C03632=1072.520,220.619,417.871,174.022,27.766,154.945
C03633=1072.515,220.371,417.896,174.019,27.761,154.944
C03634=1072.509,220.122,417.922,174.017,27.758,154.944
C03635=1072.503,219.873,417.948,174.015,27.754,154.943
C03636=1072.497,219.625,417.973,174.012,27.750,154.943
C03637=1072.491,219.377,417.999,174.010,27.746,154.942
C03638=1072.485,219.128,418.025,174.009,27.743,154.941
C03639=1072.479,218.879,418.050,174.006,27.738,154.941
C03640=1072.473,218.630,418.076,174.004,27.734,154.940
C03641=1072.468,218.382,418.101,174.002,27.731,154.940
C03642=1072.462,218.133,418.127,173.999,27.727,154.939
C03643=1072.456,217.885,418.152,173.998,27.723,154.938
C03644=1072.450,217.636,418.178,173.996,27.719,154.938
C03645=1072.444,217.387,418.204,173.994,27.715,154.937
C03646=1072.439,217.139,418.229,173.991,27.711,154.936
C03647=1072.433,216.890,418.254,173.989,27.707,154.936
C03648=1072.427,216.641,418.280,173.987,27.703,154.935
C03649=1072.421,216.393,418.305,173.985,27.699,154.935
C03650=1072.415,216.144,418.331,173.983,27.695,154.934
C03651=1072.410,215.896,418.356,173.981,27.692,154.933
C03652=1072.404,215.647,418.382,173.978,27.688,154.933
C03653=1072.398,215.398,418.407,173.976,27.684,154.932
C03654=1072.392,215.149,418.433,173.975,27.680,154.931
C03655=1072.386,214.901,418.458,173.972,27.676,154.931
C03656=1072.381,214.652,418.482,173.970,27.672,154.930
C03657=1072.375,214.403,418.508,173.968,27.668,154.930
C03658=1072.369,214.154,418.534,173.965,27.664,154.929
C03659=1072.363,213.906,418.559,173.964,27.660,154.928
C03660=1072.358,213.657,418.585,173.962,27.656,154.928
C03661=1072.352,213.409,418.610,173.960,27.652,154.927
C03662=1072.346,213.161,418.635,173.957,27.648,154.926
C03663=1072.340,212.912,418.660,173.956,27.645,154.926
C03664=1072.335,212.663,418.685,173.954,27.641,154.925
C03665=1072.328,212.414,418.711,173.951,27.637,154.925
C03666=1072.323,212.166,418.736,173.949,27.633,154.924
C03667=1072.317,211.917,418.760,173.947,27.629,154.923
C03668=1072.311,211.668,418.786,173.945,27.625,154.923
C03669=1072.306,211.420,418.811,173.943,27.621,154.922
C03670=1072.300,211.171,418.837,173.941,27.617,154.922
C03671=1072.294,210.922,418.861,173.939,27.613,154.921
C03672=1072.288,210.673,418.887,173.937,27.609,154.920
C03673=1072.282,210.425,418.912,173.935,27.606,154.920
C03674=1072.276,210.176,418.936,173.933,27.602,154.919
C03675=1072.270,209.927,418.962,173.930,27.598,154.918
C03676=1072.264,209.679,418.987,173.928,27.593,154.918
C03677=1072.258,209.430,419.011,173.927,27.590,154.917
C03678=1072.249,209.010,419.054,173.923,27.583,154.916
C03679=1072.239,208.591,419.096,173.919,27.577,154.915
C03680=1072.229,208.171,419.138,173.916,27.570,154.914
C03681=1072.220,207.751,419.180,173.912,27.563,154.913
C03682=1072.195,206.710,419.281,173.782,27.496,154.911
C03683=1072.190,206.461,419.306,173.780,27.493,154.911
C03684=1072.184,206.212,419.330,173.778,27.490,154.911
C03685=1072.178,205.964,419.354,173.776,27.487,154.910
C03686=1072.173,205.715,419.378,173.773,27.484,154.910
C03687=1072.167,205.466,419.403,173.771,27.480,154.909
C03688=1072.161,205.217,419.427,173.769,27.477,154.909
C03689=1072.155,204.969,419.451,173.767,27.475,154.909
C03690=1072.150,204.720,419.475,173.765,27.472,154.908
C03691=1072.144,204.471,419.500,173.762,27.469,154.908
C03692=1072.139,204.222,419.524,173.760,27.465,154.907
C03693=1072.133,203.974,419.548,173.758,27.463,154.907
C03694=1072.127,203.724,419.572,173.756,27.460,154.907
C03695=1072.122,203.476,419.596,173.753,27.457,154.906
C03696=1072.116,203.227,419.619,173.751,27.454,154.906
C03697=1072.111,202.979,419.644,173.749,27.451,154.905
C03698=1072.105,202.729,419.668,173.747,27.448,154.905
C03699=1072.099,202.481,419.693,173.745,27.444,154.905
C03700=1072.094,202.232,419.716,173.742,27.441,154.904
C03701=1072.088,201.983,419.740,173.741,27.439,154.904
C03702=1072.082,201.734,419.764,173.738,27.436,154.903
C03703=1072.076,201.486,419.788,173.736,27.433,154.903
C03704=1072.070,201.238,419.812,173.733,27.430,154.903
C03705=1072.065,200.988,419.836,173.732,27.427,154.902
C03706=1072.059,200.739,419.859,173.729,27.424,154.902
C03707=1072.053,200.491,419.883,173.727,27.421,154.902
C03708=1072.047,200.241,419.907,173.724,27.418,154.901
C03709=1072.041,199.993,419.931,173.723,27.416,154.901
C03710=1072.036,199.744,419.955,173.720,27.413,154.900
C03711=1072.030,199.495,419.978,173.718,27.410,154.900
C03712=1072.024,199.246,420.002,173.716,27.407,154.900
C03713=1072.018,198.998,420.026,173.714,27.404,154.899
C03714=1072.013,198.749,420.050,173.712,27.401,154.899
C03715=1072.007,198.500,420.073,173.709,27.398,154.898
C03716=1072.001,198.251,420.097,173.707,27.395,154.898
C03717=1071.996,198.002,420.121,173.705,27.393,154.898
C03718=1071.989,197.754,420.144,173.703,27.390,154.897
C03719=1071.984,197.505,420.168,173.700,27.387,154.897
C03720=1071.978,197.256,420.192,173.699,27.384,154.897
C03721=1071.972,197.007,420.216,173.696,27.381,154.896
C03722=1071.967,196.758,420.239,173.694,27.378,154.896
C03723=1071.961,196.510,420.263,173.692,27.375,154.895
C03724=1071.956,196.261,420.286,173.690,27.372,154.895
C03725=1071.950,196.012,420.310,173.688,27.369,154.895
C03726=1071.943,195.763,420.333,173.685,27.366,154.894
C03727=1071.938,195.514,420.358,173.684,27.364,154.894
C03728=1071.932,195.265,420.381,173.681,27.361,154.893
C03729=1071.927,195.017,420.405,173.679,27.358,154.893
C03730=1071.921,194.768,420.428,173.677,27.355,154.893
C03731=1071.915,194.520,420.451,173.675,27.352,154.892
C03732=1071.910,194.270,420.475,173.672,27.349,154.892
C03733=1071.904,194.021,420.499,173.671,27.346,154.892
C03734=1071.898,193.773,420.522,173.668,27.343,154.891
C03735=1071.893,193.523,420.546,173.666,27.340,154.891
C03736=1071.887,193.275,420.569,173.664,27.337,154.890
C03737=1071.881,193.026,420.592,173.662,27.334,154.890
C03738=1071.876,192.778,420.616,173.660,27.331,154.890
C03739=1071.870,192.529,420.639,173.658,27.328,154.889
C03740=1071.864,192.280,420.662,173.656,27.325,154.889
C03741=1071.859,192.031,420.687,173.653,27.323,154.888
C03742=1071.853,191.782,420.709,173.652,27.320,154.888
C03743=1071.847,191.501,420.736,173.649,27.317,154.888
C03744=1071.841,191.219,420.762,173.647,27.314,154.887
C03745=1071.834,190.938,420.789,173.645,27.310,154.887
C03746=1071.828,190.656,420.816,173.642,27.307,154.886
C03747=1071.822,190.407,420.839,173.640,27.304,154.886
C03748=1071.817,190.158,420.862,173.637,27.301,154.886
C03749=1071.811,189.909,420.885,173.636,27.298,154.885
C03750=1071.805,189.661,420.909,173.633,27.295,154.885
C03751=1071.800,189.411,420.932,173.631,27.292,154.884
C03752=1071.795,189.162,420.955,173.629,27.289,154.884
C03753=1071.789,188.914,420.978,173.627,27.286,154.884
C03754=1071.783,188.665,421.002,173.625,27.283,154.883
C03755=1071.778,188.416,421.025,173.623,27.281,154.883
C03756=1071.772,188.167,421.048,173.621,27.278,154.882
C03757=1071.766,187.918,421.071,173.619,27.275,154.882
C03758=1071.761,187.669,421.095,173.617,27.272,154.882
C03759=1071.755,187.421,421.119,173.614,27.269,154.881
C03760=1071.750,187.172,421.141,173.613,27.267,154.881
C03761=1071.744,186.923,421.164,173.610,27.263,154.881
C03762=1071.739,186.674,421.188,173.608,27.260,154.880
C03763=1071.733,186.425,421.211,173.606,27.258,154.880
C03764=1071.728,186.176,421.234,173.604,27.255,154.879
C03765=1071.722,185.927,421.257,173.602,27.252,154.879
C03766=1071.717,185.678,421.280,173.600,27.249,154.879
C03767=1071.711,185.429,421.303,173.598,27.246,154.878
C03768=1071.705,185.180,421.326,173.596,27.243,154.878
C03769=1071.700,184.931,421.349,173.594,27.240,154.877
C03770=1071.694,184.683,421.372,173.592,27.237,154.877
C03771=1071.688,184.433,421.395,173.590,27.234,154.877
C03772=1071.682,184.185,421.418,173.587,27.232,154.876
C03773=1071.677,183.936,421.441,173.586,27.229,154.876
C03774=1071.671,183.687,421.464,173.583,27.226,154.875
C03775=1071.665,183.438,421.487,173.582,27.224,154.875
C03776=1071.659,183.189,421.510,173.579,27.221,154.875
C03777=1071.653,182.940,421.532,173.577,27.218,154.874
C03778=1071.647,182.691,421.555,173.575,27.215,154.874
C03779=1071.642,182.443,421.578,173.573,27.212,154.874
C03780=1071.636,182.194,421.601,173.571,27.210,154.873
C03781=1071.630,181.945,421.624,173.569,27.207,154.873
C03782=1071.624,181.696,421.646,173.567,27.204,154.873
C03783=1071.618,181.447,421.669,173.565,27.201,154.872
C03784=1071.612,181.198,421.691,173.563,27.198,154.872
C03785=1071.607,180.949,421.714,173.561,27.196,154.872
C03786=1071.602,180.701,421.737,173.559,27.193,154.871
C03787=1071.595,180.452,421.759,173.557,27.190,154.871
C03788=1071.589,180.203,421.782,173.555,27.188,154.871
C03789=1071.584,179.954,421.805,173.552,27.185,154.870
C03790=1071.578,179.705,421.827,173.551,27.182,154.870
C03791=1071.573,179.456,421.850,173.548,27.179,154.869
C03792=1071.566,179.207,421.873,173.547,27.177,154.869
C03793=1071.560,178.958,421.896,173.544,27.174,154.869
C03794=1071.555,178.709,421.919,173.543,27.171,154.868
C03795=1071.549,178.460,421.941,173.540,27.168,154.868
C03796=1071.543,178.211,421.963,173.539,27.166,154.868
C03797=1071.537,177.962,421.986,173.536,27.163,154.867
C03798=1071.532,177.714,422.008,173.534,27.160,154.867
C03799=1071.526,177.465,422.031,173.532,27.157,154.867
C03800=1071.520,177.216,422.053,173.530,27.154,154.866
C03801=1071.514,176.967,422.076,173.529,27.152,154.866
C03802=1071.509,176.718,422.098,173.526,27.148,154.865
C03803=1071.503,176.469,422.121,173.525,27.146,154.865
C03804=1071.497,176.220,422.144,173.522,27.143,154.865
C03805=1071.492,175.971,422.166,173.521,27.140,154.864
C03806=1071.486,175.723,422.189,173.518,27.137,154.864
C03807=1071.479,175.441,422.214,173.516,27.134,154.864
C03808=1071.473,175.158,422.239,173.513,27.131,154.863
C03809=1071.466,174.877,422.265,173.512,27.129,154.863
C03810=1071.460,174.595,422.290,173.510,27.125,154.862
C03811=1071.454,174.345,422.312,173.507,27.122,154.862
C03812=1071.448,174.096,422.335,173.506,27.120,154.862
C03813=1071.444,173.847,422.357,173.503,27.117,154.861
C03814=1071.437,173.599,422.380,173.502,27.114,154.861
C03815=1071.431,173.350,422.403,173.499,27.111,154.861
C03816=1071.426,173.100,422.425,173.498,27.109,154.860
C03817=1071.420,172.852,422.447,173.495,27.106,154.860
C03818=1071.415,172.603,422.469,173.494,27.103,154.859
C03819=1071.409,172.354,422.492,173.491,27.100,154.859
C03820=1071.403,172.105,422.514,173.490,27.097,154.859
C03821=1071.398,171.857,422.536,173.488,27.094,154.858
C03822=1071.392,171.607,422.558,173.486,27.092,154.858
C03823=1071.386,171.359,422.581,173.484,27.089,154.858
C03824=1071.380,171.109,422.603,173.482,27.086,154.857
C03825=1071.375,170.860,422.625,173.480,27.083,154.857
C03826=1071.369,170.612,422.647,173.478,27.081,154.856
C03827=1071.364,170.362,422.669,173.476,27.078,154.856
C03828=1071.358,170.113,422.692,173.474,27.075,154.856
C03829=1071.352,169.865,422.714,173.472,27.072,154.855
C03830=1071.347,169.616,422.737,173.470,27.069,154.855
C03831=1071.341,169.366,422.759,173.468,27.066,154.855
C03832=1071.336,169.118,422.780,173.466,27.064,154.854
C03833=1071.330,168.869,422.803,173.464,27.061,154.854
C03834=1071.324,168.619,422.825,173.463,27.058,154.853
C03835=1071.319,168.371,422.846,173.460,27.055,154.853
C03836=1071.313,168.122,422.869,173.459,27.052,154.853
C03837=1071.308,167.872,422.892,173.456,27.050,154.852
C03838=1071.302,167.624,422.913,173.455,27.047,154.852
C03839=1071.296,167.375,422.936,173.452,27.044,154.852
C03840=1071.290,167.126,422.958,173.451,27.041,154.851
C03841=1071.285,166.877,422.979,173.448,27.038,154.851
C03842=1071.280,166.628,423.002,173.447,27.036,154.851
C03843=1071.274,166.380,423.024,173.445,27.033,154.850
C03844=1071.269,166.130,423.046,173.443,27.030,154.850
C03845=1071.263,165.881,423.067,173.442,27.027,154.849
C03846=1071.258,165.632,423.089,173.439,27.024,154.849
C03847=1071.252,165.383,423.112,173.438,27.022,154.849
C03848=1071.246,165.135,423.134,173.435,27.019,154.848
C03849=1071.241,164.885,423.156,173.434,27.016,154.848
C03850=1071.235,164.636,423.177,173.431,27.013,154.848
C03851=1071.230,164.387,423.199,173.430,27.010,154.847
C03852=1071.224,164.138,423.222,173.428,27.008,154.847
C03853=1071.219,163.890,423.243,173.426,27.005,154.846
C03854=1071.213,163.640,423.266,173.424,27.002,154.846
C03855=1071.208,163.392,423.287,173.422,26.999,154.846
C03856=1071.202,163.142,423.309,173.421,26.997,154.845
C03857=1071.197,162.894,423.330,173.418,26.994,154.845
C03858=1071.191,162.645,423.353,173.417,26.991,154.844
C03859=1071.186,162.395,423.376,173.415,26.988,154.844
C03860=1071.180,162.147,423.397,173.413,26.985,154.844
C03861=1071.175,161.897,423.419,173.411,26.983,154.843
C03862=1071.169,161.649,423.440,173.409,26.980,154.843
C03863=1071.164,161.399,423.463,173.407,26.977,154.843
C03864=1071.158,161.151,423.484,173.405,26.974,154.842
C03865=1071.152,160.902,423.506,173.403,26.972,154.842
C03866=1071.147,160.653,423.527,173.402,26.969,154.841
C03867=1071.141,160.404,423.549,173.400,26.966,154.841
C03868=1071.135,160.154,423.571,173.398,26.963,154.841
C03869=1071.129,159.906,423.592,173.396,26.960,154.840
C03870=1071.124,159.656,423.614,173.394,26.958,154.840
C03871=1071.117,159.374,423.639,173.392,26.955,154.840
C03872=1071.111,159.092,423.663,173.389,26.951,154.839
C03873=1071.104,158.810,423.687,173.388,26.949,154.839
C03874=1071.098,158.527,423.711,173.386,26.946,154.838
C03875=1071.092,158.278,423.734,173.384,26.943,154.838
C03876=1071.087,158.029,423.755,173.382,26.940,154.838
C03877=1071.080,157.780,423.776,173.380,26.937,154.837
C03878=1071.075,157.531,423.798,173.378,26.934,154.837
C03879=1071.069,157.282,423.820,173.376,26.932,154.837
C03880=1071.064,157.033,423.841,173.375,26.929,154.836
C03881=1071.058,156.784,423.863,173.372,26.926,154.836
C03882=1071.052,156.535,423.883,173.371,26.924,154.836
C03883=1071.046,156.286,423.905,173.369,26.920,154.835
C03884=1071.042,156.037,423.927,173.367,26.918,154.835
C03885=1071.035,155.788,423.949,173.366,26.915,154.834
C03886=1071.030,155.539,423.970,173.363,26.912,154.834
C03887=1071.024,155.290,423.991,173.362,26.910,154.834
C03888=1071.018,155.041,424.012,173.359,26.907,154.833
C03889=1071.012,154.792,424.034,173.358,26.904,154.833
C03890=1071.007,154.543,424.055,173.356,26.902,154.833
C03891=1071.000,154.294,424.077,173.354,26.899,154.832
C03892=1070.996,154.045,424.098,173.352,26.896,154.832
C03893=1070.990,153.795,424.119,173.351,26.893,154.832
C03894=1070.984,153.547,424.141,173.348,26.891,154.831
C03895=1070.978,153.298,424.162,173.347,26.888,154.831
C03896=1070.973,153.049,424.183,173.345,26.885,154.830
C03897=1070.967,152.799,424.204,173.343,26.883,154.830
C03898=1070.961,152.551,424.226,173.342,26.880,154.830
C03899=1070.955,152.302,424.247,173.339,26.877,154.829
C03900=1070.950,152.053,424.268,173.338,26.875,154.829
C03901=1070.944,151.804,424.289,173.336,26.872,154.829
C03902=1070.938,151.555,424.311,173.334,26.869,154.828
C03903=1070.933,151.306,424.331,173.332,26.866,154.828
C03904=1070.927,151.056,424.353,173.331,26.864,154.828
C03905=1070.921,150.808,424.374,173.328,26.861,154.827
C03906=1070.915,150.558,424.395,173.327,26.858,154.827
C03907=1070.910,150.310,424.416,173.324,26.855,154.827
C03908=1070.904,150.061,424.437,173.323,26.853,154.826
C03909=1070.898,149.811,424.459,173.322,26.850,154.826
C03910=1070.893,149.563,424.480,173.319,26.847,154.826
C03911=1070.887,149.313,424.501,173.318,26.844,154.825
C03912=1070.881,149.064,424.522,173.316,26.842,154.825
C03913=1070.876,148.815,424.543,173.314,26.839,154.824
C03914=1070.870,148.566,424.564,173.312,26.836,154.824
C03915=1070.864,148.317,424.585,173.311,26.834,154.824
C03916=1070.858,148.068,424.606,173.308,26.830,154.823
C03917=1070.853,147.819,424.627,173.307,26.828,154.823
C03918=1070.847,147.570,424.648,173.305,26.825,154.823
C03919=1070.842,147.320,424.669,173.303,26.823,154.822
C03920=1070.836,147.072,424.690,173.301,26.820,154.822
C03921=1070.829,146.822,424.711,173.300,26.817,154.821
C03922=1070.824,146.574,424.732,173.298,26.815,154.821
C03923=1070.819,146.325,424.753,173.296,26.812,154.821
C03924=1070.813,146.076,424.774,173.295,26.809,154.820
C03925=1070.807,145.826,424.795,173.292,26.807,154.820
C03926=1070.802,145.578,424.816,173.291,26.804,154.820
C03927=1070.795,145.328,424.836,173.289,26.801,154.819
C03928=1070.790,145.079,424.857,173.287,26.799,154.819
C03929=1070.784,144.830,424.879,173.285,26.796,154.819
C03930=1070.778,144.581,424.899,173.284,26.793,154.818
C03931=1070.773,144.332,424.920,173.281,26.790,154.818
C03932=1070.766,144.083,424.941,173.280,26.788,154.818
C03933=1070.761,143.834,424.961,173.279,26.785,154.817
C03934=1070.755,143.585,424.983,173.276,26.782,154.817
C03935=1070.749,143.302,425.006,173.275,26.779,154.816
C03936=1070.742,143.020,425.030,173.272,26.776,154.816
C03937=1070.736,142.737,425.053,173.271,26.773,154.816
C03938=1070.729,142.455,425.077,173.269,26.770,154.815
C03939=1070.724,142.205,425.098,173.267,26.767,154.815
C03940=1070.718,141.956,425.118,173.265,26.765,154.815
C03941=1070.712,141.707,425.139,173.263,26.762,154.814
C03942=1070.707,141.458,425.160,173.262,26.759,154.814
C03943=1070.702,141.209,425.180,173.259,26.756,154.813
C03944=1070.696,140.959,425.201,173.258,26.754,154.813
C03945=1070.689,140.711,425.222,173.256,26.751,154.813
C03946=1070.684,140.462,425.242,173.255,26.748,154.812
C03947=1070.679,140.213,425.263,173.252,26.746,154.812
C03948=1070.672,139.963,425.283,173.251,26.743,154.812
C03949=1070.667,139.715,425.305,173.250,26.740,154.811
C03950=1070.661,139.466,425.325,173.247,26.737,154.811
C03951=1070.655,139.216,425.345,173.246,26.735,154.811
C03952=1070.650,138.967,425.366,173.244,26.732,154.810
C03953=1070.644,138.718,425.387,173.243,26.730,154.810
C03954=1070.638,138.469,425.407,173.240,26.726,154.809
C03955=1070.632,138.220,425.428,173.239,26.724,154.809
C03956=1070.626,137.971,425.448,173.237,26.721,154.809
C03957=1070.621,137.722,425.469,173.235,26.718,154.808
C03958=1070.616,137.473,425.489,173.234,26.716,154.808
C03959=1070.609,137.223,425.510,173.232,26.713,154.808
C03960=1070.604,136.974,425.530,173.231,26.710,154.807
C03961=1070.598,136.725,425.550,173.228,26.707,154.807
C03962=1070.593,136.476,425.571,173.227,26.705,154.807
C03963=1070.586,136.227,425.592,173.225,26.702,154.806
C03964=1070.580,135.978,425.612,173.223,26.699,154.806
C03965=1070.575,135.729,425.633,173.221,26.697,154.806
C03966=1070.569,135.480,425.653,173.220,26.694,154.805
C03967=1070.564,135.231,425.673,173.218,26.691,154.805
C03968=1070.557,134.982,425.694,173.216,26.689,154.805
C03969=1070.552,134.733,425.714,173.215,26.686,154.804
C03970=1070.546,134.484,425.734,173.213,26.683,154.804
C03971=1070.541,134.235,425.755,173.212,26.681,154.803
C03972=1070.535,133.986,425.775,173.209,26.678,154.803
C03973=1070.529,133.736,425.796,173.208,26.675,154.803
C03974=1070.523,133.487,425.815,173.206,26.673,154.802
C03975=1070.518,133.238,425.836,173.205,26.670,154.802
C03976=1070.512,132.989,425.856,173.202,26.667,154.802
C03977=1070.506,132.740,425.877,173.201,26.665,154.801
C03978=1070.500,132.491,425.897,173.199,26.662,154.801
C03979=1070.495,132.242,425.917,173.198,26.659,154.800
C03980=1070.489,131.992,425.937,173.196,26.656,154.800
C03981=1070.484,131.743,425.957,173.194,26.654,154.800
C03982=1070.478,131.494,425.977,173.193,26.651,154.799
C03983=1070.472,131.245,425.997,173.191,26.649,154.799
C03984=1070.466,130.996,426.018,173.189,26.646,154.799
C03985=1070.460,130.747,426.038,173.187,26.643,154.798
C03986=1070.454,130.498,426.058,173.186,26.640,154.798
C03987=1070.448,130.249,426.078,173.184,26.638,154.798
C03988=1070.443,129.999,426.098,173.182,26.635,154.797
C03989=1070.437,129.751,426.118,173.180,26.632,154.797
C03990=1070.430,129.501,426.138,173.179,26.630,154.797
C03991=1070.424,129.252,426.158,173.178,26.627,154.796
C03992=1070.419,129.003,426.179,173.175,26.624,154.796
C03993=1070.413,128.754,426.198,173.174,26.622,154.796
C03994=1070.407,128.505,426.218,173.172,26.619,154.795
C03995=1070.401,128.256,426.238,173.171,26.617,154.795
C03996=1070.396,128.006,426.259,173.168,26.614,154.795
C03997=1070.390,127.757,426.279,173.167,26.611,154.794
C03998=1070.384,127.508,426.298,173.165,26.609,154.794
C03999=1070.378,127.226,426.321,173.163,26.606,154.793
C04000=1070.371,126.943,426.344,173.162,26.602,154.793
C04001=1070.364,126.660,426.366,173.159,26.599,154.793
C04002=1070.358,126.377,426.389,173.158,26.596,154.792
C04003=1070.352,126.128,426.409,173.156,26.594,154.792
C04004=1070.346,125.879,426.428,173.154,26.591,154.792
C04005=1070.340,125.630,426.448,173.153,26.588,154.791
C04006=1070.335,125.380,426.468,173.151,26.586,154.791
C04007=1070.329,125.132,426.488,173.150,26.583,154.790
C04008=1070.323,124.883,426.508,173.148,26.580,154.790
C04009=1070.317,124.633,426.527,173.146,26.578,154.790
C04010=1070.311,124.385,426.547,173.144,26.575,154.789
C04011=1070.306,124.134,426.568,173.143,26.572,154.789
C04012=1070.300,123.885,426.588,173.141,26.570,154.789
C04013=1070.294,123.636,426.608,173.140,26.567,154.788
C04014=1070.288,123.387,426.627,173.138,26.564,154.788
C04015=1070.282,123.138,426.647,173.136,26.562,154.788
C04016=1070.277,122.888,426.667,173.135,26.559,154.787
C04017=1070.271,122.640,426.687,173.133,26.556,154.787
C04018=1070.265,122.391,426.706,173.131,26.553,154.787
C04019=1070.260,122.141,426.726,173.129,26.551,154.786
C04020=1070.254,121.893,426.746,173.128,26.548,154.786
C04021=1070.248,121.643,426.765,173.126,26.545,154.785
C04022=1070.243,121.394,426.785,173.125,26.543,154.785
C04023=1070.237,121.145,426.805,173.123,26.540,154.785
C04024=1070.231,120.896,426.825,173.121,26.537,154.784
C04025=1070.225,120.646,426.844,173.120,26.534,154.784
C04026=1070.219,120.398,426.864,173.118,26.532,154.784
C04027=1070.214,120.148,426.883,173.117,26.529,154.783
C04028=1070.208,119.899,426.904,173.115,26.526,154.783
C04029=1070.203,119.650,426.923,173.113,26.523,154.782
C04030=1070.197,119.401,426.943,173.112,26.521,154.782
C04031=1070.191,119.151,426.962,173.110,26.518,154.782
C04032=1070.185,118.903,426.982,173.109,26.516,154.781
C04033=1070.180,118.654,427.001,173.107,26.513,154.781
C04034=1070.174,118.405,427.021,173.105,26.510,154.781
C04035=1070.168,118.156,427.040,173.103,26.507,154.780
C04036=1070.163,117.906,427.060,173.102,26.505,154.780
C04037=1070.157,117.657,427.080,173.100,26.502,154.780
C04038=1070.151,117.408,427.099,173.099,26.499,154.779
C04039=1070.146,117.159,427.119,173.098,26.496,154.779
C04040=1070.140,116.909,427.138,173.095,26.493,154.778
C04041=1070.134,116.660,427.158,173.094,26.491,154.778
C04042=1070.128,116.411,427.178,173.092,26.488,154.778
C04043=1070.122,116.162,427.197,173.091,26.485,154.777
C04044=1070.117,115.912,427.217,173.090,26.482,154.777
C04045=1070.112,115.664,427.236,173.087,26.480,154.777
C04046=1070.106,115.414,427.256,173.086,26.477,154.776
C04047=1070.101,115.165,427.275,173.084,26.474,154.776
C04048=1070.095,114.916,427.295,173.083,26.471,154.775
C04049=1070.089,114.667,427.314,173.081,26.469,154.775
C04050=1070.083,114.417,427.333,173.080,26.466,154.775
C04051=1070.077,114.168,427.353,173.078,26.463,154.774
C04052=1070.072,113.919,427.372,173.076,26.460,154.774
C04053=1070.067,113.670,427.391,173.075,26.458,154.774
C04054=1070.061,113.421,427.411,173.073,26.455,154.773
C04055=1070.055,113.172,427.431,173.072,26.452,154.773
C04056=1070.049,112.923,427.450,173.070,26.450,154.773
C04057=1070.043,112.673,427.468,173.069,26.447,154.772
C04058=1070.037,112.424,427.488,173.066,26.444,154.772
C04059=1070.031,112.175,427.507,173.065,26.442,154.771
C04060=1070.025,111.926,427.527,173.064,26.439,154.771
C04061=1070.020,111.676,427.546,173.062,26.436,154.771
C04062=1070.015,111.428,427.565,173.061,26.433,154.770
C04063=1070.007,111.144,427.587,173.058,26.430,154.770
C04064=1070.001,110.861,427.609,173.057,26.427,154.769
C04065=1069.995,110.579,427.630,173.055,26.424,154.769
C04066=1069.988,110.297,427.652,173.053,26.421,154.769
C04067=1069.982,110.047,427.671,173.052,26.419,154.768
C04068=1069.976,109.798,427.691,173.050,26.416,154.768
C04069=1069.970,109.549,427.709,173.048,26.413,154.768
C04070=1069.964,109.299,427.728,173.047,26.410,154.767
C04071=1069.959,109.050,427.748,173.045,26.408,154.767
C04072=1069.953,108.800,427.767,173.044,26.405,154.767
C04073=1069.946,108.551,427.786,173.042,26.402,154.766
C04074=1069.941,108.303,427.804,173.041,26.400,154.766
C04075=1069.936,108.053,427.824,173.039,26.397,154.765
C04076=1069.930,107.804,427.843,173.037,26.394,154.765
C04077=1069.924,107.555,427.862,173.035,26.392,154.765
C04078=1069.918,107.305,427.881,173.034,26.389,154.764
C04079=1069.912,107.056,427.900,173.033,26.386,154.764
C04080=1069.906,106.807,427.918,173.031,26.383,154.764
C04081=1069.901,106.558,427.938,173.030,26.381,154.763
C04082=1069.895,106.308,427.957,173.028,26.378,154.763
C04083=1069.889,106.059,427.976,173.026,26.375,154.763
C04084=1069.883,105.810,427.995,173.024,26.373,154.762
C04085=1069.878,105.561,428.014,173.023,26.370,154.762
C04086=1069.872,105.312,428.033,173.022,26.367,154.761
C04087=1069.866,105.063,428.052,173.020,26.364,154.761
C04088=1069.860,104.813,428.071,173.019,26.362,154.761
C04089=1069.854,104.564,428.090,173.017,26.359,154.760
C04090=1069.848,104.315,428.108,173.016,26.356,154.760
C04091=1069.843,104.066,428.128,173.013,26.354,154.760
C04092=1069.837,103.816,428.147,173.012,26.351,154.759
C04093=1069.831,103.567,428.165,173.011,26.348,154.759
C04094=1069.826,103.319,428.184,173.009,26.345,154.758
C04095=1069.820,103.069,428.204,173.008,26.343,154.758
C04096=1069.814,102.820,428.223,173.006,26.340,154.758
C04097=1069.808,102.570,428.241,173.005,26.337,154.757
C04098=1069.803,102.321,428.260,173.004,26.335,154.757
C04099=1069.797,102.072,428.279,173.001,26.332,154.757
C04100=1069.791,101.823,428.298,173.000,26.329,154.756
C04101=1069.786,101.574,428.316,172.998,26.326,154.756
C04102=1069.779,101.325,428.335,172.997,26.324,154.755
C04103=1069.774,101.075,428.354,172.995,26.321,154.755
C04104=1069.768,100.825,428.373,172.994,26.318,154.755
C04105=1069.762,100.577,428.391,172.993,26.316,154.754
C04106=1069.757,100.328,428.410,172.991,26.313,154.754
C04107=1069.750,100.078,428.429,172.989,26.310,154.754
C04108=1069.744,99.829,428.447,172.987,26.307,154.753
C04109=1069.739,99.580,428.466,172.986,26.305,154.753
C04110=1069.733,99.331,428.484,172.984,26.302,154.753
C04111=1069.727,99.081,428.504,172.983,26.299,154.752
C04112=1069.721,98.832,428.522,172.982,26.297,154.752
C04113=1069.716,98.583,428.541,172.980,26.294,154.752
C04114=1069.709,98.334,428.559,172.979,26.291,154.751
C04115=1069.704,98.084,428.578,172.977,26.289,154.751
C04116=1069.698,97.835,428.596,172.975,26.286,154.751
C04117=1069.692,97.586,428.615,172.974,26.283,154.750
C04118=1069.686,97.337,428.634,172.972,26.281,154.750
C04119=1069.680,97.087,428.652,172.971,26.278,154.749
C04120=1069.675,96.838,428.671,172.969,26.275,154.749
C04121=1069.668,96.589,428.689,172.968,26.272,154.749
C04122=1069.663,96.339,428.708,172.966,26.270,154.748
C04123=1069.657,96.091,428.726,172.965,26.267,154.748
C04124=1069.651,95.842,428.745,172.964,26.264,154.748
C04125=1069.645,95.591,428.763,172.962,26.262,154.747
C04126=1069.640,95.343,428.782,172.960,26.259,154.747
C04127=1069.633,95.060,428.802,172.958,26.256,154.746
C04128=1069.627,94.777,428.824,172.957,26.253,154.746
C04129=1069.620,94.494,428.844,172.955,26.250,154.746
C04130=1069.613,94.211,428.866,172.953,26.247,154.745
C04131=1069.608,93.963,428.884,172.952,26.244,154.745
C04132=1069.602,93.713,428.902,172.950,26.242,154.744
C04133=1069.596,93.464,428.921,172.949,26.239,154.744
C04134=1069.590,93.215,428.939,172.948,26.236,154.744
C04135=1069.585,92.965,428.958,172.945,26.233,154.743
C04136=1069.579,92.716,428.976,172.944,26.231,154.743
C04137=1069.573,92.467,428.994,172.942,26.228,154.743
C04138=1069.567,92.217,429.013,172.941,26.225,154.742
C04139=1069.561,91.969,429.031,172.940,26.222,154.742
C04140=1069.556,91.719,429.049,172.938,26.220,154.742
C04141=1069.550,91.470,429.068,172.937,26.217,154.741
C04142=1069.544,91.220,429.086,172.935,26.214,154.741
C04143=1069.538,90.971,429.105,172.934,26.211,154.740
C04144=1069.533,90.722,429.122,172.932,26.209,154.740
C04145=1069.527,90.473,429.141,172.931,26.206,154.740
C04146=1069.520,90.223,429.159,172.929,26.203,154.739
C04147=1069.515,89.975,429.177,172.927,26.201,154.739
C04148=1069.509,89.725,429.196,172.926,26.198,154.739
C04149=1069.504,89.476,429.213,172.924,26.195,154.738
C04150=1069.497,89.226,429.232,172.923,26.193,154.738
C04151=1069.491,88.977,429.250,172.922,26.190,154.737
C04152=1069.485,88.728,429.268,172.920,26.187,154.737
C04153=1069.479,88.479,429.286,172.919,26.185,154.737
C04154=1069.474,88.229,429.304,172.917,26.182,154.736
C04155=1069.468,87.980,429.323,172.916,26.179,154.736
C04156=1069.462,87.730,429.341,172.914,26.177,154.736
C04157=1069.456,87.481,429.359,172.913,26.174,154.735
C04158=1069.450,87.232,429.377,172.911,26.171,154.735
C04159=1069.444,86.983,429.395,172.909,26.168,154.735
C04160=1069.438,86.733,429.413,172.908,26.166,154.734
C04161=1069.432,86.485,429.431,172.906,26.163,154.734
C04162=1069.427,86.235,429.449,172.905,26.160,154.733
C04163=1069.421,85.985,429.467,172.904,26.158,154.733
C04164=1069.415,85.737,429.486,172.902,26.155,154.733
C04165=1069.409,85.487,429.504,172.901,26.152,154.732
C04166=1069.403,85.238,429.521,172.899,26.150,154.732
C04167=1069.397,84.988,429.539,172.898,26.147,154.732
C04168=1069.392,84.740,429.557,172.897,26.144,154.731
C04169=1069.385,84.490,429.575,172.895,26.141,154.731
C04170=1069.380,84.241,429.593,172.894,26.139,154.731
C04171=1069.375,83.991,429.611,172.892,26.136,154.730
C04172=1069.369,83.743,429.630,172.890,26.133,154.730
C04173=1069.363,83.493,429.648,172.888,26.130,154.730
C04174=1069.357,83.244,429.665,172.887,26.128,154.729
C04175=1069.351,82.994,429.683,172.886,26.125,154.729
C04176=1069.345,82.745,429.701,172.884,26.122,154.728
C04177=1069.339,82.496,429.719,172.883,26.120,154.728
C04178=1069.333,82.247,429.737,172.881,26.117,154.728
C04179=1069.327,81.997,429.755,172.880,26.114,154.727
C04180=1069.322,81.748,429.772,172.879,26.111,154.727
C04181=1069.316,81.498,429.790,172.877,26.109,154.727
C04182=1069.310,81.249,429.808,172.876,26.106,154.726
C04183=1069.304,81.000,429.827,172.874,26.103,154.726
C04184=1069.298,80.751,429.844,172.873,26.100,154.725
C04185=1069.293,80.502,429.862,172.872,26.098,154.725
C04186=1069.287,80.252,429.880,172.870,26.095,154.725
C04187=1069.282,80.003,429.898,172.869,26.092,154.724
C04188=1069.276,79.753,429.916,172.867,26.089,154.724
C04189=1069.270,79.504,429.933,172.865,26.087,154.724
C04190=1069.264,79.254,429.951,172.864,26.084,154.723
C04191=1069.258,78.972,429.971,172.862,26.081,154.723
C04192=1069.251,78.689,429.992,172.861,26.078,154.722
C04193=1069.245,78.407,430.011,172.859,26.074,154.722
C04194=1069.238,78.124,430.031,172.857,26.072,154.722
C04195=1069.232,77.875,430.049,172.856,26.069,154.721
C04196=1069.226,77.625,430.067,172.855,26.066,154.721
C04197=1069.220,77.376,430.084,172.853,26.064,154.720
C04198=1069.214,77.126,430.102,172.852,26.061,154.720
C04199=1069.209,76.877,430.120,172.850,26.058,154.720
C04200=1069.202,76.628,430.137,172.849,26.056,154.719
C04201=1069.196,76.379,430.155,172.847,26.053,154.719
C04202=1069.191,76.130,430.172,172.846,26.050,154.719
C04203=1069.185,75.880,430.190,172.845,26.048,154.718
C04204=1069.179,75.631,430.208,172.842,26.044,154.718
C04205=1069.173,75.381,430.226,172.841,26.042,154.717
C04206=1069.167,75.132,430.243,172.839,26.039,154.717
C04207=1069.161,74.883,430.260,172.838,26.036,154.717
C04208=1069.155,74.634,430.278,172.837,26.034,154.716
C04209=1069.150,74.385,430.296,172.835,26.031,154.716
C04210=1069.144,74.135,430.314,172.834,26.028,154.716
C04211=1069.138,73.886,430.331,172.832,26.026,154.715
C04212=1069.132,73.636,430.348,172.831,26.023,154.715
C04213=1069.126,73.387,430.366,172.830,26.020,154.715
C04214=1069.120,73.138,430.383,172.828,26.018,154.714
C04215=1069.114,72.888,430.401,172.827,26.015,154.714
C04216=1069.109,72.639,430.419,172.825,26.012,154.713
C04217=1069.103,72.390,430.436,172.824,26.010,154.713
C04218=1069.096,72.140,430.453,172.823,26.007,154.713
C04219=1069.091,71.891,430.470,172.821,26.004,154.712
C04220=1069.086,71.642,430.488,172.820,26.001,154.712
C04221=1069.079,71.392,430.505,172.818,25.999,154.712
C04222=1069.073,71.143,430.523,172.817,25.996,154.711
C04223=1069.068,70.894,430.540,172.816,25.993,154.711
C04224=1069.062,70.644,430.558,172.814,25.991,154.711
C04225=1069.056,70.395,430.575,172.813,25.988,154.710
C04226=1069.050,70.146,430.592,172.810,25.985,154.710
C04227=1069.044,69.896,430.610,172.809,25.982,154.709
C04228=1069.039,69.647,430.627,172.808,25.979,154.709
C04229=1069.033,69.398,430.644,172.806,25.977,154.709
C04230=1069.026,69.148,430.662,172.805,25.974,154.708
C04231=1069.021,68.899,430.679,172.803,25.971,154.708
C04232=1069.015,68.650,430.696,172.802,25.969,154.708
C04233=1069.009,68.400,430.714,172.801,25.966,154.707
C04234=1069.003,68.151,430.731,172.799,25.963,154.707
C04235=1068.997,67.902,430.747,172.798,25.961,154.707
C04236=1068.991,67.652,430.765,172.796,25.958,154.706
C04237=1068.985,67.403,430.782,172.795,25.955,154.706
C04238=1068.980,67.154,430.800,172.794,25.952,154.705
C04239=1068.974,66.905,430.817,172.792,25.950,154.705
C04240=1068.967,66.655,430.834,172.791,25.947,154.705
C04241=1068.962,66.405,430.851,172.789,25.944,154.704
C04242=1068.956,66.157,430.868,172.788,25.942,154.704
C04243=1068.950,65.907,430.886,172.787,25.939,154.704
C04244=1068.945,65.657,430.903,172.785,25.936,154.703
C04245=1068.938,65.409,430.920,172.784,25.934,154.703
C04246=1068.933,65.160,430.937,172.782,25.931,154.703
C04247=1068.926,64.910,430.954,172.781,25.928,154.702
C04248=1068.921,64.660,430.971,172.780,25.926,154.702
C04249=1068.915,64.411,430.988,172.778,25.923,154.701
C04250=1068.909,64.161,431.006,172.777,25.920,154.701
C04251=1068.903,63.912,431.022,172.775,25.917,154.701
C04252=1068.897,63.663,431.039,172.774,25.915,154.700
C04253=1068.890,63.414,431.057,172.773,25.912,154.700
C04254=1068.884,63.164,431.073,172.770,25.909,154.700
C04255=1068.878,62.881,431.092,172.769,25.906,154.699
C04256=1068.871,62.598,431.112,172.768,25.903,154.699
C04257=1068.864,62.316,431.130,172.766,25.901,154.699
C04258=1068.857,62.032,431.150,172.764,25.897,154.698
C04259=1068.851,61.784,431.167,172.763,25.894,154.698
C04260=1068.846,61.534,431.184,172.761,25.892,154.697
C04261=1068.839,61.285,431.201,172.760,25.889,154.697
C04262=1068.833,61.035,431.217,172.758,25.886,154.697
C04263=1068.828,60.786,431.235,172.757,25.884,154.696
C04264=1068.822,60.537,431.251,172.755,25.881,154.696
C04265=1068.815,60.287,431.269,172.754,25.879,154.696
C04266=1068.810,60.038,431.285,172.753,25.876,154.695
C04267=1068.803,59.789,431.302,172.751,25.873,154.695
C04268=1068.797,59.540,431.318,172.750,25.871,154.695
C04269=1068.792,59.289,431.336,172.748,25.868,154.694
C04270=1068.785,59.041,431.353,172.747,25.865,154.694
C04271=1068.779,58.791,431.369,172.746,25.863,154.694
C04272=1068.774,58.542,431.386,172.744,25.860,154.693
C04273=1068.767,58.292,431.403,172.743,25.858,154.693
C04274=1068.761,58.043,431.419,172.741,25.855,154.692
C04275=1068.756,57.794,431.437,172.740,25.852,154.692
C04276=1068.750,57.544,431.453,172.739,25.850,154.692
C04277=1068.744,57.295,431.469,172.737,25.847,154.691
C04278=1068.738,57.045,431.487,172.736,25.844,154.691
C04279=1068.732,56.796,431.504,172.734,25.842,154.691
C04280=1068.726,56.547,431.520,172.733,25.839,154.690
C04281=1068.720,56.298,431.537,172.732,25.836,154.690
C04282=1068.714,56.048,431.554,172.730,25.834,154.690
C04283=1068.708,55.799,431.570,172.729,25.831,154.689
C04284=1068.702,55.549,431.587,172.728,25.828,154.689
C04285=1068.696,55.300,431.604,172.726,25.825,154.689
C04286=1068.690,55.050,431.620,172.725,25.823,154.688
C04287=1068.684,54.801,431.637,172.723,25.820,154.688
C04288=1068.678,54.552,431.654,172.722,25.817,154.687
C04289=1068.673,54.303,431.670,172.721,25.815,154.687
C04290=1068.667,54.053,431.687,172.719,25.812,154.687
C04291=1068.660,53.803,431.703,172.718,25.809,154.686
C04292=1068.655,53.554,431.721,172.715,25.806,154.686
C04293=1068.649,53.305,431.737,172.714,25.803,154.686
C04294=1068.643,53.056,431.753,172.713,25.801,154.685
C04295=1068.637,52.806,431.770,172.711,25.798,154.685
C04296=1068.632,52.557,431.786,172.710,25.795,154.685
C04297=1068.626,52.308,431.803,172.708,25.793,154.684
C04298=1068.620,52.058,431.820,172.707,25.790,154.684
C04299=1068.614,51.809,431.836,172.706,25.787,154.683
C04300=1068.608,51.559,431.853,172.704,25.785,154.683
C04301=1068.602,51.309,431.869,172.703,25.782,154.683
C04302=1068.596,51.060,431.886,172.702,25.779,154.682
C04303=1068.590,50.811,431.903,172.700,25.777,154.682
C04304=1068.585,50.562,431.920,172.699,25.774,154.682
C04305=1068.579,50.312,431.936,172.697,25.771,154.681
C04306=1068.573,50.063,431.952,172.696,25.768,154.681
C04307=1068.567,49.814,431.968,172.695,25.766,154.681
C04308=1068.561,49.564,431.985,172.693,25.763,154.680
C04309=1068.556,49.315,432.001,172.692,25.760,154.680
C04310=1068.550,49.065,432.018,172.690,25.758,154.680
C04311=1068.544,48.816,432.034,172.689,25.755,154.679
C04312=1068.537,48.567,432.051,172.688,25.752,154.679
C04313=1068.531,48.318,432.067,172.686,25.750,154.678
C04314=1068.526,48.068,432.084,172.685,25.747,154.678
C04315=1068.520,47.819,432.100,172.683,25.744,154.678
C04316=1068.514,47.569,432.117,172.682,25.741,154.677
C04317=1068.508,47.320,432.133,172.681,25.739,154.677
C04318=1068.502,47.071,432.149,172.679,25.736,154.677
C04319=1068.496,46.787,432.168,172.678,25.733,154.676
C04320=1068.490,46.504,432.187,172.677,25.730,154.676
C04321=1068.483,46.221,432.205,172.675,25.726,154.675
C04322=1068.477,45.938,432.223,172.673,25.723,154.675
C04323=1068.471,45.688,432.240,172.672,25.721,154.675
C04324=1068.465,45.439,432.256,172.670,25.718,154.674
C04325=1068.459,45.190,432.272,172.669,25.715,154.674
C04326=1068.453,44.940,432.288,172.668,25.712,154.673
C04327=1068.448,44.691,432.305,172.666,25.710,154.673
C04328=1068.442,44.441,432.321,172.665,25.707,154.673
C04329=1068.436,44.192,432.338,172.664,25.704,154.672
C04330=1068.430,43.943,432.354,172.662,25.702,154.672
C04331=1068.424,43.693,432.370,172.661,25.699,154.672
C04332=1068.418,43.444,432.386,172.659,25.696,154.671
C04333=1068.412,43.195,432.403,172.658,25.693,154.671
C04334=1068.406,42.945,432.419,172.657,25.691,154.671
C04335=1068.401,42.695,432.434,172.655,25.688,154.670
C04336=1068.395,42.446,432.451,172.654,25.685,154.670
C04337=1068.389,42.197,432.467,172.652,25.683,154.670
C04338=1068.383,41.947,432.483,172.651,25.680,154.669
C04339=1068.377,41.698,432.499,172.650,25.677,154.669
C04340=1068.371,41.449,432.516,172.648,25.675,154.668
C04341=1068.365,41.199,432.532,172.647,25.672,154.668
C04342=1068.359,40.949,432.548,172.645,25.670,154.668
C04343=1068.353,40.700,432.564,172.644,25.667,154.667
C04344=1068.347,40.450,432.580,172.643,25.664,154.667
C04345=1068.341,40.201,432.596,172.641,25.662,154.667
C04346=1068.335,39.952,432.613,172.640,25.659,154.666
C04347=1068.330,39.703,432.628,172.639,25.656,154.666
C04348=1068.324,39.453,432.644,172.637,25.654,154.666
C04349=1068.318,39.204,432.660,172.636,25.651,154.665
C04350=1068.312,38.955,432.676,172.634,25.648,154.665
C04351=1068.306,38.705,432.691,172.633,25.645,154.665
C04352=1068.300,38.455,432.708,172.632,25.643,154.664
C04353=1068.294,38.206,432.724,172.630,25.640,154.664
C04354=1068.288,37.957,432.740,172.629,25.637,154.663
C04355=1068.283,37.707,432.756,172.628,25.634,154.663
C04356=1068.277,37.457,432.772,172.626,25.632,154.663
C04357=1068.270,37.208,432.788,172.625,25.629,154.662
C04358=1068.264,36.958,432.803,172.623,25.627,154.662
C04359=1068.258,36.709,432.819,172.622,25.624,154.662
C04360=1068.253,36.460,432.835,172.620,25.622,154.661
C04361=1068.246,36.211,432.851,172.619,25.619,154.661
C04362=1068.241,35.961,432.867,172.618,25.616,154.661
C04363=1068.235,35.712,432.883,172.616,25.614,154.660
C04364=1068.229,35.462,432.898,172.615,25.611,154.660
C04365=1068.222,35.213,432.914,172.614,25.608,154.660
C04366=1068.216,34.964,432.930,172.612,25.606,154.659
C04367=1068.211,34.714,432.946,172.611,25.603,154.659
C04368=1068.205,34.464,432.962,172.609,25.600,154.659
C04369=1068.198,34.215,432.978,172.608,25.597,154.658
C04370=1068.193,33.966,432.993,172.607,25.595,154.658
C04371=1068.187,33.717,433.009,172.605,25.592,154.658
C04372=1068.181,33.467,433.025,172.604,25.590,154.657
C04373=1068.175,33.218,433.040,172.603,25.587,154.657
C04374=1068.169,32.968,433.057,172.601,25.585,154.657
C04375=1068.163,32.718,433.072,172.600,25.582,154.656
C04376=1068.157,32.469,433.088,172.598,25.579,154.656
C04377=1068.151,32.219,433.103,172.597,25.577,154.656
C04378=1068.146,31.971,433.119,172.596,25.574,154.655
C04379=1068.139,31.721,433.134,172.594,25.571,154.655
C04380=1068.133,31.472,433.150,172.593,25.568,154.654
C04381=1068.128,31.222,433.166,172.591,25.566,154.654
C04382=1068.122,30.972,433.182,172.590,25.563,154.654
C04383=1068.115,30.689,433.200,172.588,25.560,154.653
C04384=1068.108,30.406,433.218,172.586,25.557,154.653
C04385=1068.102,30.123,433.235,172.585,25.554,154.653
C04386=1068.095,29.840,433.253,172.584,25.551,154.652
C04387=1068.088,29.591,433.269,172.582,25.548,154.652
C04388=1068.083,29.341,433.284,172.581,25.546,154.652
C04389=1068.078,29.092,433.299,172.580,25.543,154.651
C04390=1068.071,28.843,433.315,172.578,25.540,154.651
C04391=1068.065,28.593,433.331,172.577,25.538,154.651
C04392=1068.059,28.344,433.346,172.576,25.535,154.650
C04393=1068.053,28.094,433.362,172.574,25.533,154.650
C04394=1068.048,27.845,433.378,172.573,25.530,154.649
C04395=1068.041,27.595,433.393,172.571,25.528,154.649
C04396=1068.036,27.345,433.408,172.570,25.525,154.649
C04397=1068.029,27.096,433.424,172.569,25.522,154.648
C04398=1068.023,26.846,433.439,172.567,25.519,154.648
C04399=1068.017,26.597,433.454,172.566,25.517,154.648
C04400=1068.012,26.348,433.470,172.564,25.514,154.647
C04401=1068.005,26.098,433.485,172.563,25.512,154.647
C04402=1067.999,25.849,433.501,172.562,25.509,154.647
C04403=1067.993,25.599,433.516,172.560,25.507,154.646
C04404=1067.988,25.350,433.531,172.559,25.504,154.646
C04405=1067.981,25.100,433.546,172.557,25.501,154.646
C04406=1067.975,24.851,433.563,172.556,25.498,154.645
C04407=1067.969,24.601,433.578,172.555,25.496,154.645
C04408=1067.964,24.352,433.593,172.553,25.493,154.645
C04409=1067.957,24.103,433.608,172.552,25.491,154.644
C04410=1067.952,23.853,433.624,172.551,25.488,154.644
C04411=1067.945,23.603,433.639,172.549,25.486,154.644
C04412=1067.939,23.354,433.654,172.548,25.483,154.643
C04413=1067.934,23.105,433.670,172.546,25.480,154.643
C04414=1067.927,22.855,433.685,172.545,25.478,154.643
C04415=1067.922,22.606,433.700,172.544,25.475,154.642
C04416=1067.916,22.357,433.715,172.542,25.472,154.642
C04417=1067.910,22.107,433.731,172.541,25.470,154.642
C04418=1067.903,21.858,433.746,172.539,25.467,154.641
C04419=1067.898,21.608,433.761,172.538,25.465,154.641
C04420=1067.892,21.359,433.776,172.537,25.462,154.641
C04421=1067.886,21.109,433.792,172.535,25.460,154.640
C04422=1067.880,20.860,433.807,172.534,25.457,154.640
C04423=1067.874,20.611,433.822,172.532,25.454,154.640
C04424=1067.868,20.361,433.837,172.531,25.451,154.639
C04425=1067.862,20.111,433.852,172.530,25.449,154.639
C04426=1067.857,19.862,433.868,172.528,25.447,154.639
C04427=1067.850,19.612,433.883,172.527,25.444,154.638
C04428=1067.844,19.363,433.898,172.525,25.441,154.638
C04429=1067.838,19.113,433.914,172.524,25.439,154.638
C04430=1067.832,18.864,433.928,172.523,25.436,154.637
C04431=1067.826,18.615,433.943,172.521,25.433,154.637
C04432=1067.820,18.365,433.959,172.520,25.431,154.637
C04433=1067.814,18.116,433.973,172.519,25.428,154.636
C04434=1067.808,17.866,433.988,172.517,25.426,154.636
C04435=1067.802,17.616,434.003,172.516,25.423,154.636
C04436=1067.797,17.367,434.018,172.514,25.421,154.635
C04437=1067.790,17.117,434.033,172.513,25.418,154.635
C04438=1067.784,16.868,434.049,172.512,25.415,154.635
C04439=1067.779,16.619,434.064,172.510,25.413,154.634
C04440=1067.772,16.369,434.079,172.509,25.410,154.634
C04441=1067.766,16.120,434.094,172.507,25.408,154.634
C04442=1067.761,15.870,434.109,172.506,25.405,154.633
C04443=1067.754,15.621,434.124,172.505,25.402,154.633
C04444=1067.749,15.372,434.139,172.503,25.400,154.633
C04445=1067.742,15.122,434.154,172.502,25.397,154.632
C04446=1067.737,14.872,434.169,172.500,25.395,154.632
C04447=1067.730,14.591,434.186,172.498,25.392,154.632
C04448=1067.724,14.309,434.202,172.497,25.389,154.631
C04449=1067.716,14.027,434.220,172.496,25.386,154.631
C04450=1067.710,13.745,434.236,172.494,25.383,154.631
C04451=1067.703,13.495,434.251,172.493,25.381,154.630
C04452=1067.698,13.246,434.266,172.491,25.378,154.630
C04453=1067.691,12.997,434.281,172.490,25.375,154.630
C04454=1067.685,12.747,434.296,172.489,25.373,154.629
C04455=1067.679,12.498,434.310,172.487,25.371,154.629
C04456=1067.673,12.248,434.325,172.486,25.368,154.629
C04457=1067.667,11.998,434.340,172.484,25.365,154.628
C04458=1067.661,11.749,434.354,172.483,25.363,154.628
C04459=1067.654,11.500,434.369,172.481,25.360,154.628
C04460=1067.649,11.251,434.384,172.479,25.357,154.628
C04461=1067.642,11.001,434.399,172.478,25.355,154.627
C04462=1067.636,10.751,434.414,172.476,25.353,154.627
C04463=1067.631,10.502,434.429,172.475,25.350,154.627
C04464=1067.624,10.252,434.444,172.474,25.348,154.626
C04465=1067.619,10.003,434.458,172.472,25.345,154.626
C04466=1067.613,9.753,434.473,172.471,25.342,154.626
C04467=1067.606,9.503,434.488,172.469,25.340,154.625
C04468=1067.600,9.255,434.502,172.468,25.338,154.625
C04469=1067.594,9.005,434.517,172.467,25.335,154.625
C04470=1067.588,8.755,434.531,172.465,25.332,154.624
C04471=1067.582,8.506,434.546,172.464,25.330,154.624
C04472=1067.576,8.256,434.561,172.462,25.327,154.624
C04473=1067.570,8.007,434.575,172.461,25.325,154.624
C04474=1067.564,7.757,434.590,172.460,25.322,154.623
C04475=1067.558,7.508,434.604,172.458,25.319,154.623
C04476=1067.552,7.258,434.619,172.457,25.317,154.623
C04477=1067.546,7.009,434.634,172.455,25.315,154.622
C04478=1067.540,6.760,434.649,172.454,25.312,154.622
C04479=1067.534,6.510,434.663,172.453,25.310,154.622
C04480=1067.528,6.260,434.677,172.451,25.307,154.621
C04481=1067.522,6.011,434.692,172.450,25.304,154.621
C04482=1067.516,5.761,434.706,172.448,25.302,154.621
C04483=1067.510,5.512,434.721,172.447,25.300,154.620
C04484=1067.504,5.262,434.736,172.446,25.297,154.620
C04485=1067.498,5.014,434.750,172.444,25.294,154.620
C04486=1067.492,4.763,434.765,172.443,25.292,154.620
C04487=1067.486,4.514,434.779,172.442,25.289,154.619
C04488=1067.480,4.265,434.794,172.440,25.287,154.619
C04489=1067.474,4.015,434.808,172.439,25.284,154.619
C04490=1067.468,3.765,434.823,172.437,25.282,154.618
C04491=1067.462,3.516,434.837,172.436,25.279,154.618
C04492=1067.456,3.266,434.852,172.434,25.277,154.618
C04493=1067.450,3.017,434.866,172.433,25.274,154.617
C04494=1067.444,2.767,434.881,172.432,25.272,154.617
C04495=1067.438,2.518,434.895,172.430,25.269,154.617
C04496=1067.432,2.268,434.910,172.429,25.267,154.616
C04497=1067.426,2.019,434.924,172.428,25.264,154.616
C04498=1067.420,1.769,434.939,172.426,25.262,154.616
C04499=1067.415,1.520,434.953,172.425,25.259,154.615
C04500=1067.408,1.270,434.968,172.423,25.256,154.615
C04501=1067.403,1.020,434.982,172.422,25.254,154.615
C04502=1067.397,0.771,434.996,172.420,25.252,154.615
C04503=1067.391,0.522,435.011,172.419,25.249,154.614
C04504=1067.385,0.272,435.025,172.418,25.246,154.614
C04505=1067.379,0.022,435.040,172.416,25.244,154.614
C04506=1067.373,-0.227,435.054,172.415,25.242,154.613
C04507=1067.367,-0.476,435.068,172.414,25.239,154.613
C04508=1067.361,-0.726,435.083,172.412,25.236,154.613
C04509=1067.356,-0.975,435.097,172.411,25.234,154.612
C04510=1067.349,-1.225,435.111,172.409,25.231,154.612
C04511=1067.342,-1.505,435.127,172.408,25.229,154.612
C04512=1067.335,-1.785,435.143,172.407,25.226,154.611
C04513=1067.329,-2.065,435.159,172.404,25.223,154.611
C04514=1067.322,-2.344,435.175,172.403,25.220,154.611
C04515=1067.317,-2.594,435.189,172.402,25.217,154.610
C04516=1067.311,-2.843,435.204,172.400,25.215,154.610
C04517=1067.305,-3.093,435.218,172.399,25.213,154.610
C04518=1067.299,-3.342,435.232,172.398,25.210,154.609
C04519=1067.293,-3.592,435.247,172.396,25.207,154.609
C04520=1067.287,-3.842,435.260,172.395,25.205,154.609
C04521=1067.281,-4.091,435.275,172.393,25.203,154.609
C04522=1067.275,-4.341,435.289,172.392,25.200,154.608
C04523=1067.268,-4.590,435.303,172.390,25.198,154.608
C04524=1067.262,-4.840,435.317,172.389,25.196,154.608
C04525=1067.257,-5.089,435.331,172.388,25.193,154.607
C04526=1067.250,-5.338,435.345,172.386,25.190,154.607
C04527=1067.244,-5.588,435.359,172.385,25.188,154.607
C04528=1067.239,-5.838,435.373,172.383,25.186,154.607
C04529=1067.232,-6.087,435.387,172.382,25.183,154.606
C04530=1067.226,-6.337,435.401,172.380,25.181,154.606
C04531=1067.221,-6.586,435.415,172.379,25.179,154.606
C04532=1067.214,-6.836,435.429,172.378,25.176,154.605
C04533=1067.208,-7.085,435.443,172.376,25.173,154.605
C04534=1067.202,-7.336,435.457,172.375,25.171,154.605
C04535=1067.196,-7.584,435.471,172.373,25.169,154.604
C04536=1067.190,-7.834,435.485,172.372,25.166,154.604
C04537=1067.184,-8.084,435.499,172.371,25.164,154.604
C04538=1067.178,-8.333,435.513,172.369,25.161,154.604
C04539=1067.172,-8.582,435.527,172.368,25.159,154.603
C04540=1067.166,-8.833,435.542,172.366,25.157,154.603
C04541=1067.160,-9.082,435.555,172.365,25.154,154.603
C04542=1067.154,-9.331,435.569,172.364,25.151,154.602
C04543=1067.147,-9.581,435.583,172.362,25.149,154.602
C04544=1067.142,-9.830,435.597,172.361,25.147,154.602
C04545=1067.136,-10.080,435.611,172.359,25.144,154.602
C04546=1067.129,-10.330,435.624,172.358,25.142,154.601
C04547=1067.124,-10.579,435.638,172.356,25.140,154.601
C04548=1067.117,-10.828,435.652,172.355,25.137,154.601
C04549=1067.112,-11.078,435.666,172.354,25.134,154.600
C04550=1067.106,-11.328,435.680,172.352,25.132,154.600
C04551=1067.100,-11.577,435.694,172.350,25.129,154.600
C04552=1067.094,-11.827,435.708,172.349,25.127,154.600
C04553=1067.087,-12.077,435.721,172.347,25.125,154.599
C04554=1067.081,-12.326,435.736,172.346,25.122,154.599
C04555=1067.076,-12.575,435.750,172.344,25.120,154.599
C04556=1067.070,-12.825,435.763,172.343,25.118,154.599
C04557=1067.064,-13.075,435.777,172.341,25.115,154.598
C04558=1067.057,-13.324,435.790,172.340,25.113,154.598
C04559=1067.052,-13.574,435.804,172.339,25.111,154.598
C04560=1067.047,-13.823,435.818,172.337,25.108,154.597
C04561=1067.040,-14.073,435.832,172.336,25.105,154.597
C04562=1067.034,-14.323,435.846,172.334,25.103,154.597
C04563=1067.028,-14.571,435.860,172.333,25.100,154.597
C04564=1067.022,-14.821,435.873,172.332,25.098,154.596
C04565=1067.015,-15.071,435.887,172.330,25.096,154.596
C04566=1067.010,-15.321,435.901,172.329,25.093,154.596
C04567=1067.004,-15.570,435.914,172.327,25.091,154.595
C04568=1066.998,-15.819,435.928,172.326,25.089,154.595
C04569=1066.991,-16.069,435.942,172.324,25.086,154.595
C04570=1066.985,-16.319,435.955,172.323,25.084,154.595
C04571=1066.980,-16.568,435.969,172.322,25.082,154.594
C04572=1066.974,-16.817,435.982,172.320,25.079,154.594
C04573=1066.967,-17.067,435.996,172.319,25.077,154.594
C04574=1066.961,-17.317,436.010,172.317,25.075,154.594
C04575=1066.956,-17.544,436.022,172.316,25.073,154.593
C04576=1066.950,-17.771,436.034,172.314,25.070,154.593
C04577=1066.945,-17.998,436.046,172.313,25.068,154.593
C04578=1066.939,-18.226,436.059,172.312,25.067,154.593
C04579=1066.933,-18.452,436.071,172.311,25.064,154.592
C04580=1066.928,-18.680,436.083,172.309,25.062,154.592
C04581=1066.922,-18.906,436.095,172.308,25.060,154.592
C04582=1066.917,-19.133,436.107,172.306,25.058,154.592
C04583=1066.911,-19.383,436.122,172.305,25.055,154.591
C04584=1066.905,-19.633,436.135,172.304,25.053,154.591
C04585=1066.899,-19.882,436.148,172.302,25.051,154.591
C04586=1066.893,-20.132,436.162,172.301,25.048,154.591
C04587=1066.885,-20.454,436.179,172.298,25.045,154.590
C04588=1066.877,-20.778,436.197,172.297,25.043,154.590
C04589=1066.869,-21.102,436.215,172.295,25.039,154.590
C04590=1066.861,-21.425,436.231,172.294,25.036,154.589
C04591=1066.855,-21.674,436.245,172.292,25.034,154.589
C04592=1066.850,-21.924,436.259,172.291,25.032,154.589
C04593=1066.844,-22.173,436.271,172.289,25.029,154.588
C04594=1066.837,-22.423,436.284,172.287,25.027,154.588
C04595=1066.832,-22.672,436.298,172.286,25.024,154.588
C04596=1066.825,-22.922,436.312,172.284,25.022,154.588
C04597=1066.819,-23.172,436.325,172.283,25.020,154.588
C04598=1066.814,-23.422,436.338,172.281,25.018,154.587
C04599=1066.807,-23.671,436.352,172.280,25.015,154.587
C04600=1066.801,-23.920,436.365,172.278,25.013,154.587
C04601=1066.796,-24.170,436.379,172.277,25.011,154.586
C04602=1066.790,-24.419,436.392,172.275,25.008,154.586
C04603=1066.784,-24.669,436.405,172.274,25.006,154.586
C04604=1066.777,-24.919,436.418,172.273,25.004,154.586
C04605=1066.771,-25.169,436.432,172.271,25.001,154.585
C04606=1066.765,-25.418,436.445,172.270,24.999,154.585
C04607=1066.759,-25.668,436.458,172.268,24.997,154.585
C04608=1066.754,-25.917,436.472,172.267,24.995,154.585
C04609=1066.748,-26.166,436.485,172.265,24.992,154.584
C04610=1066.742,-26.416,436.498,172.264,24.990,154.584
C04611=1066.735,-26.666,436.511,172.263,24.988,154.584
C04612=1066.730,-26.915,436.525,172.261,24.985,154.584
C04613=1066.724,-27.164,436.538,172.260,24.983,154.583
C04614=1066.718,-27.414,436.551,172.258,24.981,154.583
C04615=1066.711,-27.664,436.564,172.257,24.979,154.583
C04616=1066.705,-27.914,436.577,172.255,24.976,154.583
C04617=1066.699,-28.163,436.590,172.254,24.974,154.582
C04618=1066.693,-28.413,436.603,172.252,24.972,154.582
C04619=1066.687,-28.663,436.616,172.251,24.970,154.582
C04620=1066.681,-28.912,436.629,172.249,24.967,154.582
C04621=1066.674,-29.161,436.642,172.248,24.965,154.581
C04622=1066.668,-29.411,436.655,172.247,24.963,154.581
C04623=1066.662,-29.660,436.668,172.245,24.961,154.581
C04624=1066.656,-29.910,436.681,172.244,24.958,154.581
C04625=1066.651,-30.160,436.695,172.241,24.956,154.581
C04626=1066.644,-30.410,436.708,172.240,24.954,154.580
C04627=1066.638,-30.660,436.721,172.238,24.952,154.580
C04628=1066.632,-30.909,436.734,172.237,24.949,154.580
C04629=1066.626,-31.159,436.747,172.235,24.947,154.580
C04630=1066.620,-31.408,436.760,172.234,24.945,154.579
C04631=1066.614,-31.658,436.772,172.233,24.943,154.579
C04632=1066.608,-31.907,436.786,172.231,24.940,154.579
C04633=1066.601,-32.156,436.799,172.230,24.938,154.579
C04634=1066.596,-32.406,436.812,172.228,24.936,154.579
C04635=1066.589,-32.656,436.825,172.227,24.934,154.578
C04636=1066.583,-32.905,436.837,172.225,24.932,154.578
C04637=1066.577,-33.155,436.851,172.224,24.930,154.578
C04638=1066.571,-33.405,436.863,172.222,24.927,154.578
C04639=1066.564,-33.682,436.877,172.221,24.925,154.577
C04640=1066.558,-33.959,436.892,172.219,24.922,154.577
C04641=1066.551,-34.236,436.906,172.217,24.920,154.577
C04642=1066.545,-34.514,436.921,172.216,24.917,154.577
C04643=1066.539,-34.764,436.933,172.214,24.915,154.576
C04644=1066.533,-35.014,436.947,172.213,24.913,154.576
C04645=1066.527,-35.263,436.959,172.211,24.911,154.576
C04646=1066.520,-35.513,436.972,172.210,24.908,154.576
C04647=1066.515,-35.763,436.985,172.208,24.907,154.575
C04648=1066.508,-36.012,436.998,172.207,24.904,154.575
C04649=1066.502,-36.262,437.011,172.206,24.902,154.575
C04650=1066.497,-36.512,437.023,172.204,24.900,154.575
C04651=1066.490,-36.761,437.037,172.203,24.898,154.574
C04652=1066.484,-37.011,437.049,172.201,24.895,154.574
C04653=1066.479,-37.259,437.062,172.199,24.893,154.574
C04654=1066.473,-37.509,437.075,172.197,24.891,154.574
C04655=1066.467,-37.759,437.087,172.196,24.888,154.574
C04656=1066.461,-38.008,437.100,172.194,24.887,154.573
C04657=1066.454,-38.258,437.112,172.193,24.884,154.573
C04658=1066.448,-38.508,437.125,172.191,24.882,154.573
C04659=1066.442,-38.757,437.138,172.190,24.880,154.573
C04660=1066.436,-39.007,437.151,172.189,24.878,154.572
C04661=1066.430,-39.257,437.163,172.187,24.876,154.572
C04662=1066.424,-39.506,437.177,172.186,24.874,154.572
C04663=1066.417,-39.756,437.189,172.184,24.872,154.572
C04664=1066.411,-40.006,437.201,172.183,24.869,154.572
C04665=1066.405,-40.255,437.214,172.181,24.868,154.571
C04666=1066.399,-40.505,437.227,172.180,24.865,154.571
C04667=1066.393,-40.755,437.240,172.178,24.863,154.571
C04668=1066.387,-41.004,437.251,172.177,24.861,154.571
C04669=1066.381,-41.254,437.264,172.175,24.859,154.571
C04670=1066.375,-41.503,437.277,172.174,24.857,154.570
C04671=1066.369,-41.753,437.290,172.172,24.855,154.570
C04672=1066.363,-42.002,437.301,172.171,24.853,154.570
C04673=1066.357,-42.252,437.314,172.169,24.851,154.570
C04674=1066.351,-42.501,437.327,172.168,24.848,154.570
C04675=1066.345,-42.751,437.340,172.166,24.847,154.569
C04676=1066.338,-43.001,437.352,172.165,24.844,154.569
C04677=1066.332,-43.251,437.364,172.162,24.842,154.569
C04678=1066.326,-43.500,437.377,172.161,24.840,154.569
C04679=1066.320,-43.750,437.389,172.159,24.838,154.569
C04680=1066.314,-43.999,437.402,172.158,24.836,154.569
C04681=1066.308,-44.248,437.414,172.156,24.834,154.568
C04682=1066.302,-44.498,437.427,172.155,24.832,154.568
C04683=1066.296,-44.748,437.439,172.154,24.830,154.568
C04684=1066.290,-44.998,437.451,172.152,24.828,154.568
C04685=1066.284,-45.248,437.464,172.151,24.825,154.567
C04686=1066.278,-45.498,437.477,172.149,24.824,154.567
C04687=1066.272,-45.746,437.489,172.148,24.821,154.567
C04688=1066.265,-45.996,437.501,172.146,24.819,154.567
C04689=1066.260,-46.246,437.514,172.145,24.817,154.567
C04690=1066.254,-46.495,437.526,172.143,24.815,154.566
C04691=1066.247,-46.745,437.538,172.142,24.813,154.566
C04692=1066.241,-46.995,437.551,172.140,24.811,154.566
C04693=1066.236,-47.244,437.563,172.139,24.809,154.566
C04694=1066.229,-47.494,437.575,172.137,24.807,154.566
C04695=1066.223,-47.744,437.588,172.136,24.805,154.565
C04696=1066.217,-47.993,437.600,172.134,24.803,154.565
C04697=1066.211,-48.243,437.613,172.133,24.801,154.565
C04698=1066.205,-48.492,437.624,172.131,24.799,154.565
C04699=1066.199,-48.742,437.637,172.129,24.796,154.565
C04700=1066.194,-48.992,437.649,172.127,24.795,154.565
C04701=1066.187,-49.242,437.661,172.126,24.792,154.564
C04702=1066.181,-49.491,437.674,172.124,24.790,154.564
C04703=1066.175,-49.768,437.688,172.123,24.788,154.564
C04704=1066.168,-50.047,437.701,172.121,24.786,154.564
C04705=1066.161,-50.325,437.715,172.120,24.784,154.563
C04706=1066.154,-50.603,437.728,172.117,24.782,154.563
C04707=1066.148,-50.852,437.740,172.116,24.779,154.563
C04708=1066.142,-51.101,437.752,172.115,24.777,154.563
C04709=1066.136,-51.351,437.765,172.113,24.776,154.563
C04710=1066.129,-51.601,437.777,172.111,24.774,154.563
C04711=1066.123,-51.850,437.789,172.110,24.772,154.563
C04712=1066.117,-52.100,437.801,172.108,24.770,154.562
C04713=1066.111,-52.349,437.813,172.107,24.768,154.562
C04714=1066.105,-52.599,437.826,172.105,24.766,154.562
C04715=1066.098,-52.849,437.838,172.104,24.764,154.562
C04716=1066.092,-53.099,437.849,172.102,24.762,154.562
C04717=1066.086,-53.349,437.861,172.101,24.761,154.562
C04718=1066.080,-53.597,437.873,172.099,24.758,154.561
C04719=1066.073,-53.847,437.885,172.098,24.756,154.561
C04720=1066.067,-54.097,437.897,172.096,24.755,154.561
C04721=1066.061,-54.346,437.909,172.094,24.752,154.561
C04722=1066.055,-54.596,437.922,172.092,24.751,154.561
C04723=1066.049,-54.846,437.933,172.091,24.749,154.561
C04724=1066.042,-55.095,437.945,172.089,24.747,154.560
C04725=1066.036,-55.345,437.957,172.088,24.745,154.560
C04726=1066.030,-55.595,437.969,172.086,24.743,154.560
C04727=1066.024,-55.844,437.981,172.085,24.741,154.560
C04728=1066.018,-56.094,437.993,172.083,24.739,154.560
C04729=1066.011,-56.344,438.005,172.082,24.737,154.560
C04730=1066.005,-56.593,438.017,172.080,24.735,154.559
C04731=1066.000,-56.843,438.029,172.078,24.734,154.559
C04732=1065.993,-57.093,438.040,172.077,24.732,154.559
C04733=1065.987,-57.343,438.053,172.075,24.729,154.559
C04734=1065.981,-57.592,438.065,172.074,24.728,154.559
C04735=1065.975,-57.841,438.076,172.072,24.726,154.559
C04736=1065.969,-58.092,438.088,172.071,24.724,154.558
C04737=1065.962,-58.341,438.100,172.069,24.722,154.558
C04738=1065.956,-58.590,438.112,172.068,24.720,154.558
C04739=1065.950,-58.840,438.124,172.066,24.719,154.558
C04740=1065.944,-59.090,438.135,172.065,24.717,154.558
C04741=1065.938,-59.339,438.147,172.062,24.715,154.558
C04742=1065.931,-59.589,438.159,172.061,24.713,154.558
C04743=1065.926,-59.839,438.171,172.059,24.711,154.558
C04744=1065.920,-60.088,438.182,172.058,24.709,154.557
C04745=1065.913,-60.338,438.194,172.056,24.707,154.557
C04746=1065.907,-60.588,438.206,172.055,24.705,154.557
C04747=1065.901,-60.837,438.218,172.053,24.703,154.557
C04748=1065.895,-61.086,438.230,172.052,24.701,154.557
C04749=1065.889,-61.337,438.242,172.050,24.700,154.557
C04750=1065.883,-61.586,438.253,172.048,24.698,154.556
C04751=1065.877,-61.836,438.264,172.047,24.696,154.556
C04752=1065.870,-62.086,438.276,172.045,24.694,154.556
C04753=1065.865,-62.335,438.289,172.044,24.692,154.556
C04754=1065.858,-62.585,438.300,172.042,24.690,154.556
C04755=1065.852,-62.835,438.312,172.041,24.689,154.556
C04756=1065.847,-63.084,438.323,172.039,24.687,154.556
C04757=1065.840,-63.334,438.335,172.038,24.685,154.555
C04758=1065.834,-63.583,438.347,172.036,24.683,154.555
C04759=1065.828,-63.833,438.358,172.035,24.681,154.555
C04760=1065.822,-64.083,438.371,172.033,24.680,154.555
C04761=1065.816,-64.332,438.381,172.031,24.678,154.555
C04762=1065.810,-64.582,438.393,172.029,24.676,154.555
C04763=1065.804,-64.831,438.404,172.027,24.674,154.555
C04764=1065.798,-65.081,438.417,172.026,24.672,154.554
C04765=1065.792,-65.331,438.428,172.024,24.670,154.554
C04766=1065.785,-65.580,438.440,172.023,24.668,154.554
C04767=1065.779,-65.860,438.453,172.021,24.666,154.554
C04768=1065.772,-66.139,438.466,172.020,24.665,154.554
C04769=1065.766,-66.418,438.478,172.017,24.662,154.554
C04770=1065.759,-66.697,438.492,172.016,24.660,154.554
C04771=1065.753,-66.947,438.503,172.014,24.658,154.553
C04772=1065.746,-67.196,438.515,172.013,24.656,154.553
C04773=1065.740,-67.446,438.526,172.011,24.655,154.553
C04774=1065.735,-67.696,438.538,172.010,24.653,154.553
C04775=1065.728,-67.946,438.550,172.008,24.652,154.553
C04776=1065.723,-68.195,438.560,172.006,24.650,154.553
C04777=1065.716,-68.445,438.572,172.005,24.648,154.553
C04778=1065.710,-68.694,438.583,172.003,24.646,154.553
C04779=1065.704,-68.944,438.596,172.002,24.644,154.552
C04780=1065.699,-69.194,438.607,172.000,24.643,154.552
C04781=1065.692,-69.444,438.618,171.999,24.641,154.552
C04782=1065.686,-69.693,438.630,171.997,24.639,154.552
C04783=1065.680,-69.943,438.641,171.995,24.637,154.552
C04784=1065.675,-70.193,438.652,171.993,24.635,154.552
C04785=1065.668,-70.442,438.664,171.992,24.633,154.552
C04786=1065.663,-70.692,438.675,171.990,24.632,154.552
C04787=1065.657,-70.941,438.686,171.988,24.630,154.551
C04788=1065.650,-71.191,438.698,171.987,24.628,154.551
C04789=1065.645,-71.441,438.709,171.985,24.626,154.551
C04790=1065.639,-71.691,438.721,171.984,24.625,154.551
C04791=1065.633,-71.940,438.732,171.982,24.623,154.551
C04792=1065.626,-72.190,438.743,171.981,24.621,154.551
C04793=1065.621,-72.439,438.754,171.979,24.619,154.551
C04794=1065.615,-72.689,438.767,171.977,24.618,154.551
C04795=1065.609,-72.939,438.778,171.976,24.616,154.550
C04796=1065.603,-73.188,438.789,171.974,24.614,154.550
C04797=1065.597,-73.438,438.801,171.973,24.612,154.550
C04798=1065.591,-73.687,438.812,171.971,24.611,154.550
C04799=1065.585,-73.937,438.823,171.970,24.609,154.550
C04800=1065.579,-74.187,438.834,171.968,24.607,154.550
C04801=1065.572,-74.436,438.846,171.967,24.606,154.550
C04802=1065.566,-74.686,438.856,171.965,24.604,154.550
C04803=1065.560,-74.936,438.868,171.963,24.603,154.550
C04804=1065.554,-75.186,438.879,171.962,24.601,154.549
C04805=1065.548,-75.436,438.890,171.959,24.599,154.549
C04806=1065.542,-75.685,438.901,171.958,24.597,154.549
C04807=1065.536,-75.934,438.912,171.956,24.596,154.549
C04808=1065.530,-76.184,438.924,171.955,24.594,154.549
C04809=1065.524,-76.434,438.934,171.953,24.592,154.549
C04810=1065.518,-76.684,438.946,171.951,24.591,154.549
C04811=1065.512,-76.934,438.957,171.950,24.589,154.549
C04812=1065.505,-77.183,438.969,171.948,24.588,154.549
C04813=1065.500,-77.433,438.979,171.947,24.586,154.549
C04814=1065.493,-77.683,438.991,171.945,24.584,154.548
C04815=1065.488,-77.932,439.002,171.943,24.583,154.548
C04816=1065.481,-78.181,439.012,171.942,24.581,154.548
C04817=1065.475,-78.432,439.023,171.940,24.580,154.548
C04818=1065.469,-78.681,439.034,171.939,24.578,154.548
C04819=1065.463,-78.931,439.045,171.937,24.576,154.548
C04820=1065.457,-79.180,439.057,171.935,24.575,154.548
C04821=1065.451,-79.430,439.068,171.934,24.573,154.548
C04822=1065.445,-79.680,439.079,171.932,24.572,154.548
C04823=1065.439,-79.929,439.090,171.931,24.570,154.548
C04824=1065.432,-80.180,439.101,171.929,24.569,154.548
C04825=1065.426,-80.429,439.111,171.927,24.567,154.547
C04826=1065.420,-80.678,439.122,171.926,24.565,154.547
C04827=1065.414,-80.928,439.133,171.923,24.563,154.547
C04828=1065.407,-81.178,439.144,171.922,24.562,154.547
C04829=1065.401,-81.428,439.155,171.920,24.560,154.547
C04830=1065.395,-81.677,439.166,171.918,24.559,154.547
C04831=1065.388,-81.959,439.178,171.917,24.557,154.547
C04832=1065.381,-82.240,439.191,171.915,24.556,154.547
C04833=1065.374,-82.522,439.203,171.913,24.554,154.547
C04834=1065.367,-82.803,439.215,171.911,24.552,154.547
C04835=1065.361,-83.052,439.226,171.909,24.551,154.547
C04836=1065.355,-83.301,439.237,171.908,24.549,154.547
C04837=1065.349,-83.551,439.248,171.906,24.548,154.547
C04838=1065.342,-83.801,439.257,171.904,24.546,154.547
C04839=1065.337,-84.051,439.268,171.903,24.545,154.546
C04840=1065.330,-84.301,439.279,171.901,24.543,154.546
C04841=1065.324,-84.550,439.290,171.900,24.542,154.546
C04842=1065.318,-84.800,439.301,171.898,24.540,154.546
C04843=1065.312,-85.050,439.312,171.896,24.539,154.546
C04844=1065.305,-85.299,439.322,171.895,24.538,154.546
C04845=1065.299,-85.549,439.333,171.893,24.536,154.546
C04846=1065.293,-85.799,439.344,171.891,24.535,154.546
C04847=1065.287,-86.048,439.355,171.890,24.533,154.546
C04848=1065.280,-86.298,439.366,171.888,24.532,154.546
C04849=1065.275,-86.548,439.376,171.887,24.530,154.546
C04850=1065.269,-86.797,439.386,171.884,24.529,154.546
C04851=1065.262,-87.048,439.397,171.882,24.527,154.546
C04852=1065.256,-87.297,439.408,171.881,24.526,154.546
C04853=1065.250,-87.546,439.419,171.879,24.524,154.546
C04854=1065.244,-87.796,439.430,171.878,24.523,154.546
C04855=1065.238,-88.046,439.441,171.876,24.521,154.546
C04856=1065.232,-88.296,439.450,171.874,24.520,154.546
C04857=1065.226,-88.545,439.461,171.873,24.518,154.545
C04858=1065.220,-88.795,439.472,171.871,24.517,154.545
C04859=1065.213,-89.045,439.483,171.869,24.516,154.545
C04860=1065.207,-89.294,439.494,171.868,24.514,154.545
C04861=1065.202,-89.544,439.504,171.866,24.513,154.545
C04862=1065.195,-89.794,439.514,171.864,24.511,154.545
C04863=1065.189,-90.044,439.525,171.863,24.510,154.545
C04864=1065.183,-90.293,439.536,171.861,24.508,154.545
C04865=1065.177,-90.543,439.546,171.859,24.507,154.545
C04866=1065.171,-90.793,439.557,171.858,24.506,154.545
C04867=1065.164,-91.042,439.567,171.856,24.505,154.545
C04868=1065.159,-91.292,439.578,171.855,24.503,154.545
C04869=1065.153,-91.541,439.588,171.853,24.501,154.545
C04870=1065.146,-91.792,439.599,171.851,24.500,154.545
C04871=1065.140,-92.041,439.610,171.849,24.499,154.545
C04872=1065.134,-92.291,439.619,171.848,24.497,154.545
C04873=1065.129,-92.540,439.630,171.846,24.496,154.545
C04874=1065.122,-92.790,439.641,171.845,24.495,154.545
C04875=1065.116,-93.040,439.652,171.843,24.493,154.545
C04876=1065.110,-93.290,439.662,171.841,24.492,154.545
C04877=1065.104,-93.539,439.672,171.839,24.490,154.545
C04878=1065.098,-93.789,439.683,171.837,24.489,154.545
C04879=1065.092,-94.038,439.693,171.835,24.487,154.545
C04880=1065.086,-94.289,439.704,171.834,24.486,154.544
C04881=1065.080,-94.539,439.714,171.832,24.485,154.544
C04882=1065.074,-94.788,439.724,171.830,24.484,154.544
C04883=1065.068,-95.037,439.735,171.829,24.482,154.544
C04884=1065.062,-95.287,439.745,171.827,24.481,154.544
C04885=1065.056,-95.537,439.756,171.825,24.479,154.544
C04886=1065.049,-95.787,439.766,171.824,24.478,154.544
C04887=1065.044,-96.037,439.777,171.822,24.477,154.544
C04888=1065.038,-96.286,439.787,171.820,24.476,154.544
C04889=1065.032,-96.536,439.797,171.819,24.474,154.544
C04890=1065.026,-96.785,439.808,171.817,24.473,154.544
C04891=1065.020,-97.035,439.817,171.815,24.471,154.544
C04892=1065.014,-97.285,439.828,171.814,24.470,154.544
C04893=1065.007,-97.535,439.839,171.812,24.469,154.544
C04894=1065.001,-97.785,439.849,171.810,24.468,154.544
C04895=1064.994,-98.068,439.861,171.809,24.466,154.544
C04896=1064.987,-98.351,439.872,171.806,24.465,154.544
C04897=1064.980,-98.635,439.884,171.804,24.463,154.544
C04898=1064.974,-98.919,439.895,171.803,24.462,154.544
C04899=1064.967,-99.168,439.906,171.801,24.461,154.544
C04900=1064.961,-99.418,439.915,171.799,24.460,154.544
C04901=1064.955,-99.667,439.926,171.798,24.458,154.544
C04902=1064.949,-99.917,439.936,171.796,24.457,154.544
C04903=1064.942,-100.168,439.946,171.794,24.456,154.544
C04904=1064.936,-100.417,439.956,171.793,24.455,154.544
C04905=1064.930,-100.667,439.966,171.791,24.453,154.544
C04906=1064.924,-100.916,439.976,171.789,24.452,154.544
C04907=1064.918,-101.166,439.986,171.788,24.451,154.544
C04908=1064.912,-101.415,439.997,171.785,24.449,154.544
C04909=1064.906,-101.665,440.006,171.783,24.448,154.544
C04910=1064.900,-101.915,440.017,171.781,24.447,154.544
C04911=1064.893,-102.165,440.027,171.780,24.446,154.544
C04912=1064.887,-102.415,440.037,171.778,24.445,154.544
C04913=1064.881,-102.665,440.048,171.776,24.444,154.544
C04914=1064.875,-102.914,440.057,171.775,24.442,154.544
C04915=1064.869,-103.163,440.067,171.773,24.441,154.544
C04916=1064.863,-103.414,440.078,171.771,24.440,154.544
C04917=1064.857,-103.663,440.087,171.770,24.439,154.544
C04918=1064.851,-103.913,440.097,171.768,24.438,154.544
C04919=1064.844,-104.162,440.107,171.766,24.437,154.544
C04920=1064.839,-104.412,440.117,171.764,24.435,154.544
C04921=1064.832,-104.662,440.127,171.763,24.434,154.544
C04922=1064.826,-104.911,440.137,171.761,24.433,154.544
C04923=1064.820,-105.162,440.148,171.759,24.432,154.544
C04924=1064.814,-105.411,440.158,171.758,24.431,154.544
C04925=1064.808,-105.661,440.167,171.756,24.430,154.544
C04926=1064.801,-105.911,440.177,171.754,24.428,154.544
C04927=1064.796,-106.161,440.188,171.753,24.427,154.544
C04928=1064.790,-106.410,440.197,171.751,24.426,154.544
C04929=1064.783,-106.660,440.207,171.749,24.425,154.544
C04930=1064.777,-106.910,440.217,171.747,24.424,154.544
C04931=1064.771,-107.159,440.227,171.746,24.423,154.544
C04932=1064.765,-107.409,440.237,171.744,24.422,154.544
C04933=1064.759,-107.659,440.247,171.742,24.421,154.544
C04934=1064.753,-107.909,440.256,171.740,24.420,154.544
C04935=1064.746,-108.158,440.266,171.739,24.419,154.544
C04936=1064.740,-108.408,440.276,171.737,24.418,154.544
C04937=1064.734,-108.658,440.286,171.735,24.416,154.544
C04938=1064.729,-108.908,440.296,171.733,24.416,154.544
C04939=1064.723,-109.157,440.305,171.732,24.414,154.544
C04940=1064.716,-109.407,440.316,171.730,24.413,154.544
C04941=1064.710,-109.656,440.325,171.728,24.412,154.544
C04942=1064.704,-109.906,440.335,171.727,24.411,154.544
C04943=1064.698,-110.156,440.344,171.725,24.410,154.544
C04944=1064.691,-110.406,440.354,171.723,24.409,154.544
C04945=1064.685,-110.655,440.364,171.721,24.408,154.544
C04946=1064.679,-110.905,440.374,171.720,24.407,154.545
C04947=1064.673,-111.155,440.383,171.718,24.406,154.545
C04948=1064.667,-111.405,440.393,171.716,24.405,154.545
C04949=1064.661,-111.655,440.403,171.714,24.404,154.545
C04950=1064.655,-111.904,440.413,171.713,24.403,154.545
C04951=1064.649,-112.154,440.422,171.711,24.402,154.545
C04952=1064.642,-112.404,440.432,171.709,24.401,154.545
C04953=1064.636,-112.653,440.442,171.707,24.400,154.545
C04954=1064.630,-112.903,440.452,171.706,24.399,154.545
C04955=1064.624,-113.153,440.461,171.704,24.398,154.545
C04956=1064.617,-113.402,440.471,171.702,24.397,154.545
C04957=1064.611,-113.652,440.480,171.700,24.396,154.545
C04958=1064.605,-113.902,440.490,171.699,24.395,154.545
C04959=1064.599,-114.184,440.501,171.696,24.394,154.545
C04960=1064.592,-114.466,440.511,171.694,24.393,154.545
C04961=1064.584,-114.748,440.522,171.692,24.392,154.545
C04962=1064.578,-115.029,440.533,171.691,24.391,154.545
C04963=1064.572,-115.279,440.542,171.689,24.390,154.545
C04964=1064.565,-115.528,440.552,171.687,24.389,154.545
C04965=1064.559,-115.778,440.561,171.685,24.388,154.545
C04966=1064.553,-116.028,440.571,171.684,24.387,154.545
C04967=1064.547,-116.278,440.580,171.682,24.386,154.545
C04968=1064.541,-116.528,440.590,171.680,24.385,154.546
C04969=1064.535,-116.777,440.600,171.678,24.384,154.546
C04970=1064.528,-117.027,440.609,171.677,24.383,154.546
C04971=1064.522,-117.277,440.619,171.675,24.383,154.546
C04972=1064.516,-117.527,440.628,171.673,24.381,154.546
C04973=1064.510,-117.777,440.638,171.671,24.381,154.546
C04974=1064.504,-118.026,440.647,171.669,24.380,154.546
C04975=1064.498,-118.275,440.657,171.668,24.379,154.546
C04976=1064.492,-118.525,440.666,171.666,24.378,154.546
C04977=1064.486,-118.775,440.676,171.664,24.377,154.546
C04978=1064.480,-119.025,440.685,171.662,24.376,154.546
C04979=1064.473,-119.275,440.695,171.661,24.375,154.546
C04980=1064.467,-119.524,440.704,171.659,24.375,154.546
C04981=1064.460,-119.774,440.713,171.657,24.373,154.546
C04982=1064.454,-120.024,440.722,171.655,24.373,154.546
C04983=1064.448,-120.274,440.732,171.653,24.372,154.547
C04984=1064.443,-120.523,440.741,171.652,24.371,154.547
C04985=1064.437,-120.773,440.751,171.650,24.370,154.547
C04986=1064.430,-121.023,440.760,171.648,24.369,154.547
C04987=1064.424,-121.273,440.770,171.646,24.369,154.547
C04988=1064.418,-121.522,440.779,171.645,24.367,154.547
C04989=1064.411,-121.773,440.788,171.643,24.367,154.547
C04990=1064.405,-122.022,440.797,171.641,24.366,154.547
C04991=1064.400,-122.271,440.806,171.639,24.365,154.547
C04992=1064.394,-122.521,440.816,171.637,24.364,154.547
C04993=1064.387,-122.771,440.825,171.635,24.364,154.547
C04994=1064.381,-123.021,440.835,171.634,24.363,154.547
C04995=1064.375,-123.271,440.843,171.632,24.362,154.548
C04996=1064.368,-123.521,440.853,171.630,24.361,154.547
C04997=1064.363,-123.770,440.862,171.628,24.360,154.548
C04998=1064.357,-124.020,440.872,171.626,24.360,154.548
C04999=1064.351,-124.270,440.880,171.625,24.359,154.548
C05000=1064.345,-124.520,440.890,171.623,24.358,154.548
C05001=1064.338,-124.769,440.899,171.621,24.357,154.548
C05002=1064.332,-125.018,440.908,171.619,24.356,154.548
C05003=1064.326,-125.269,440.917,171.617,24.356,154.548
C05004=1064.320,-125.519,440.927,171.616,24.355,154.548
C05005=1064.313,-125.768,440.936,171.614,24.354,154.548
C05006=1064.307,-126.018,440.945,171.612,24.354,154.548
C05007=1064.301,-126.268,440.954,171.610,24.353,154.549
C05008=1064.295,-126.517,440.963,171.608,24.352,154.549
C05009=1064.289,-126.767,440.972,171.606,24.351,154.549
C05010=1064.283,-127.017,440.981,171.605,24.351,154.549
C05011=1064.277,-127.267,440.991,171.603,24.350,154.549
C05012=1064.270,-127.516,440.999,171.601,24.349,154.549
C05013=1064.264,-127.766,441.009,171.599,24.348,154.549
C05014=1064.258,-128.016,441.018,171.597,24.348,154.549
C05015=1064.255,-128.267,441.028,171.596,24.346,154.549
C05016=1064.253,-128.518,441.039,171.594,24.344,154.549
C05017=1064.252,-128.768,441.051,171.593,24.341,154.549
C05018=1064.253,-129.018,441.062,171.592,24.337,154.548
C05019=1064.255,-129.271,441.077,171.592,24.333,154.547
C05020=1064.259,-129.522,441.090,171.591,24.329,154.547
C05021=1064.265,-129.774,441.105,171.591,24.323,154.546
C05022=1064.272,-130.023,441.120,171.590,24.317,154.545
C05023=1063.888,-130.046,440.938,171.544,24.469,154.578
C05024=1063.881,-129.796,440.923,171.543,24.474,154.579
C05025=1063.875,-129.545,440.908,171.544,24.479,154.579
C05026=1063.871,-129.293,440.893,171.545,24.484,154.580
C05027=1063.869,-129.041,440.880,171.546,24.488,154.581
C05028=1063.868,-128.791,440.868,171.546,24.492,154.581
C05029=1063.869,-128.540,440.855,171.547,24.495,154.582
C05030=1063.871,-128.289,440.845,171.548,24.497,154.582
C05031=1063.875,-128.039,440.835,171.550,24.499,154.582
C05032=1063.880,-127.789,440.825,171.552,24.499,154.582
C05033=1063.885,-127.539,440.816,171.554,24.500,154.582
C05034=1063.892,-127.290,440.807,171.555,24.501,154.582
C05035=1063.899,-127.040,440.798,171.557,24.501,154.582
C05036=1063.904,-126.789,440.789,171.559,24.502,154.582
C05037=1063.911,-126.540,440.780,171.561,24.503,154.582
C05038=1063.917,-126.291,440.771,171.563,24.504,154.582
C05039=1063.923,-126.040,440.762,171.564,24.505,154.581
C05040=1063.929,-125.791,440.752,171.566,24.505,154.581
C05041=1063.936,-125.541,440.743,171.568,24.506,154.581
C05042=1063.942,-125.291,440.734,171.570,24.507,154.581
C05043=1063.947,-125.042,440.725,171.572,24.507,154.581
C05044=1063.953,-124.792,440.716,171.574,24.508,154.581
C05045=1063.960,-124.542,440.707,171.575,24.509,154.581
C05046=1063.967,-124.293,440.697,171.577,24.510,154.581
C05047=1063.972,-124.042,440.688,171.579,24.511,154.581
C05048=1063.979,-123.792,440.679,171.581,24.511,154.581
C05049=1063.984,-123.543,440.670,171.583,24.512,154.580
C05050=1063.991,-123.294,440.661,171.584,24.513,154.580
C05051=1063.997,-123.044,440.651,171.586,24.514,154.580
C05052=1064.003,-122.794,440.642,171.588,24.515,154.580
C05053=1064.009,-122.544,440.633,171.590,24.515,154.580
C05054=1064.015,-122.294,440.623,171.592,24.516,154.580
C05055=1064.021,-122.045,440.614,171.593,24.517,154.580
C05056=1064.028,-121.795,440.605,171.595,24.518,154.580
C05057=1064.034,-121.545,440.596,171.597,24.519,154.580
C05058=1064.040,-121.295,440.586,171.599,24.519,154.580
C05059=1064.046,-121.045,440.577,171.601,24.520,154.580
C05060=1064.052,-120.796,440.567,171.602,24.521,154.580
C05061=1064.058,-120.546,440.558,171.604,24.522,154.579
C05062=1064.064,-120.297,440.548,171.606,24.522,154.579
C05063=1064.070,-120.047,440.539,171.608,24.524,154.579
C05064=1064.076,-119.797,440.529,171.610,24.524,154.579
C05065=1064.083,-119.547,440.521,171.611,24.525,154.579
C05066=1064.089,-119.297,440.512,171.613,24.526,154.579
C05067=1064.095,-119.047,440.502,171.615,24.527,154.579
C05068=1064.102,-118.798,440.492,171.617,24.528,154.579
C05069=1064.108,-118.548,440.483,171.618,24.529,154.579
C05070=1064.113,-118.299,440.474,171.620,24.530,154.579
C05071=1064.119,-118.049,440.464,171.622,24.530,154.579
C05072=1064.126,-117.799,440.454,171.624,24.532,154.579
C05073=1064.132,-117.549,440.445,171.626,24.532,154.579
C05074=1064.138,-117.299,440.435,171.627,24.533,154.579
C05075=1064.144,-117.050,440.426,171.629,24.534,154.579
C05076=1064.150,-116.800,440.416,171.631,24.535,154.578
C05077=1064.156,-116.550,440.407,171.633,24.536,154.578
C05078=1064.163,-116.300,440.397,171.635,24.537,154.578
C05079=1064.170,-116.051,440.388,171.636,24.538,154.578
C05080=1064.176,-115.801,440.379,171.638,24.539,154.578
C05081=1064.182,-115.551,440.369,171.640,24.539,154.578
C05082=1064.188,-115.301,440.359,171.642,24.541,154.578
C05083=1064.194,-115.052,440.350,171.643,24.541,154.578
C05084=1064.200,-114.770,440.339,171.645,24.542,154.578
C05085=1064.208,-114.488,440.328,171.648,24.543,154.578
C05086=1064.215,-114.206,440.317,171.650,24.545,154.578
C05087=1064.221,-113.925,440.306,171.651,24.546,154.578
C05088=1064.227,-113.675,440.297,171.653,24.547,154.578
C05089=1064.233,-113.425,440.287,171.655,24.548,154.578
C05090=1064.239,-113.175,440.278,171.657,24.549,154.578
C05091=1064.245,-112.925,440.268,171.658,24.550,154.578
C05092=1064.252,-112.676,440.259,171.660,24.550,154.578
C05093=1064.258,-112.426,440.249,171.662,24.552,154.578
C05094=1064.264,-112.177,440.239,171.664,24.552,154.578
C05095=1064.270,-111.927,440.229,171.665,24.554,154.578
C05096=1064.277,-111.677,440.220,171.667,24.554,154.577
C05097=1064.283,-111.427,440.210,171.669,24.556,154.577
C05098=1064.288,-111.177,440.200,171.671,24.557,154.578
C05099=1064.294,-110.927,440.190,171.672,24.557,154.577
C05100=1064.301,-110.677,440.181,171.674,24.559,154.577
C05101=1064.307,-110.428,440.171,171.676,24.559,154.577
C05102=1064.313,-110.179,440.161,171.678,24.561,154.577
C05103=1064.319,-109.929,440.151,171.679,24.562,154.577
C05104=1064.326,-109.679,440.142,171.681,24.563,154.577
C05105=1064.332,-109.429,440.132,171.683,24.564,154.577
C05106=1064.338,-109.179,440.123,171.684,24.565,154.577
C05107=1064.344,-108.930,440.112,171.686,24.566,154.577
C05108=1064.350,-108.680,440.102,171.688,24.567,154.577
C05109=1064.356,-108.430,440.093,171.691,24.569,154.577
C05110=1064.362,-108.180,440.083,171.692,24.569,154.577
C05111=1064.369,-107.931,440.073,171.694,24.570,154.577
C05112=1064.375,-107.681,440.063,171.696,24.572,154.577
C05113=1064.381,-107.432,440.054,171.698,24.572,154.577
C05114=1064.386,-107.182,440.044,171.699,24.574,154.577
C05115=1064.393,-106.932,440.033,171.701,24.575,154.577
C05116=1064.399,-106.683,440.024,171.703,24.576,154.577
C05117=1064.405,-106.433,440.014,171.705,24.577,154.577
C05118=1064.412,-106.182,440.004,171.706,24.578,154.577
C05119=1064.418,-105.933,439.993,171.708,24.579,154.577
C05120=1064.424,-105.683,439.984,171.710,24.581,154.577
C05121=1064.430,-105.433,439.974,171.711,24.581,154.577
C05122=1064.437,-105.184,439.964,171.713,24.582,154.577
C05123=1064.442,-104.934,439.954,171.715,24.584,154.577
C05124=1064.448,-104.684,439.944,171.717,24.585,154.577
C05125=1064.455,-104.435,439.934,171.718,24.586,154.577
C05126=1064.460,-104.185,439.924,171.720,24.587,154.577
C05127=1064.466,-103.935,439.914,171.722,24.588,154.577
C05128=1064.473,-103.686,439.904,171.723,24.589,154.577
C05129=1064.479,-103.436,439.894,171.725,24.591,154.577
C05130=1064.484,-103.186,439.884,171.727,24.592,154.577
C05131=1064.491,-102.937,439.874,171.729,24.593,154.577
C05132=1064.497,-102.687,439.864,171.730,24.594,154.577
C05133=1064.503,-102.437,439.853,171.732,24.595,154.577
C05134=1064.510,-102.187,439.843,171.734,24.596,154.577
C05135=1064.516,-101.937,439.834,171.735,24.598,154.577
C05136=1064.521,-101.688,439.823,171.737,24.599,154.577
C05137=1064.528,-101.438,439.813,171.739,24.600,154.577
C05138=1064.534,-101.189,439.803,171.740,24.601,154.577
C05139=1064.540,-100.939,439.793,171.742,24.603,154.577
C05140=1064.546,-100.689,439.783,171.744,24.604,154.577
C05141=1064.553,-100.439,439.773,171.746,24.605,154.577
C05142=1064.558,-100.189,439.763,171.747,24.606,154.577
C05143=1064.565,-99.940,439.752,171.749,24.607,154.577
C05144=1064.571,-99.690,439.743,171.751,24.608,154.577
C05145=1064.577,-99.440,439.732,171.752,24.609,154.577
C05146=1064.583,-99.191,439.722,171.754,24.611,154.577
C05147=1064.589,-98.941,439.712,171.756,24.612,154.577
C05148=1064.596,-98.657,439.700,171.758,24.614,154.577
C05149=1064.603,-98.374,439.688,171.760,24.615,154.577
C05150=1064.611,-98.089,439.677,171.762,24.617,154.577
C05151=1064.617,-97.806,439.665,171.764,24.618,154.577
C05152=1064.623,-97.556,439.655,171.766,24.619,154.577
C05153=1064.630,-97.307,439.645,171.768,24.621,154.577
C05154=1064.635,-97.057,439.635,171.769,24.622,154.577
C05155=1064.641,-96.808,439.624,171.771,24.623,154.577
C05156=1064.648,-96.557,439.614,171.773,24.624,154.577
C05157=1064.653,-96.308,439.603,171.774,24.626,154.577
C05158=1064.660,-96.058,439.593,171.776,24.627,154.577
C05159=1064.665,-95.808,439.583,171.778,24.628,154.577
C05160=1064.672,-95.559,439.572,171.779,24.630,154.577
C05161=1064.677,-95.309,439.562,171.781,24.631,154.577
C05162=1064.684,-95.059,439.552,171.783,24.632,154.577
C05163=1064.690,-94.810,439.541,171.784,24.634,154.577
C05164=1064.695,-94.560,439.531,171.786,24.635,154.577
C05165=1064.702,-94.310,439.520,171.788,24.636,154.577
C05166=1064.708,-94.061,439.509,171.789,24.638,154.577
C05167=1064.714,-93.811,439.500,171.791,24.639,154.577
C05168=1064.720,-93.561,439.489,171.793,24.640,154.577
C05169=1064.726,-93.311,439.478,171.794,24.642,154.577
C05170=1064.732,-93.062,439.468,171.796,24.643,154.578
C05171=1064.738,-92.812,439.457,171.798,24.645,154.578
C05172=1064.744,-92.563,439.447,171.799,24.646,154.578
C05173=1064.750,-92.312,439.436,171.801,24.647,154.578
C05174=1064.757,-92.063,439.426,171.803,24.649,154.578
C05175=1064.763,-91.813,439.415,171.804,24.650,154.578
C05176=1064.768,-91.563,439.405,171.807,24.652,154.578
C05177=1064.774,-91.314,439.395,171.809,24.653,154.578
C05178=1064.781,-91.064,439.384,171.810,24.654,154.578
C05179=1064.787,-90.814,439.373,171.812,24.656,154.578
C05180=1064.793,-90.565,439.363,171.813,24.657,154.578
C05181=1064.798,-90.315,439.352,171.815,24.659,154.578
C05182=1064.806,-90.065,439.342,171.817,24.660,154.578
C05183=1064.811,-89.816,439.331,171.819,24.661,154.578
C05184=1064.817,-89.566,439.321,171.820,24.663,154.578
C05185=1064.823,-89.317,439.310,171.822,24.664,154.578
C05186=1064.830,-89.066,439.299,171.823,24.666,154.578
C05187=1064.835,-88.817,439.288,171.825,24.667,154.578
C05188=1064.842,-88.568,439.278,171.827,24.669,154.578
C05189=1064.848,-88.317,439.267,171.828,24.670,154.578
C05190=1064.854,-88.068,439.257,171.830,24.671,154.578
C05191=1064.860,-87.818,439.246,171.832,24.673,154.579
C05192=1064.866,-87.568,439.235,171.833,24.674,154.579
C05193=1064.873,-87.319,439.225,171.835,24.675,154.579
C05194=1064.879,-87.069,439.214,171.837,24.677,154.579
C05195=1064.884,-86.820,439.203,171.838,24.678,154.579
C05196=1064.891,-86.569,439.193,171.840,24.680,154.579
C05197=1064.897,-86.320,439.182,171.841,24.682,154.579
C05198=1064.903,-86.070,439.171,171.843,24.683,154.579
C05199=1064.910,-85.820,439.161,171.845,24.684,154.579
C05200=1064.915,-85.571,439.150,171.846,24.686,154.579
C05201=1064.921,-85.321,439.139,171.849,24.687,154.579
C05202=1064.928,-85.072,439.128,171.851,24.689,154.579
C05203=1064.934,-84.822,439.117,171.852,24.690,154.579
C05204=1064.940,-84.573,439.106,171.854,24.692,154.579
C05205=1064.947,-84.323,439.096,171.856,24.694,154.579
C05206=1064.952,-84.073,439.085,171.857,24.695,154.579
C05207=1064.959,-83.822,439.074,171.859,24.696,154.579
C05208=1064.964,-83.573,439.064,171.860,24.698,154.580
C05209=1064.971,-83.324,439.053,171.862,24.699,154.580
C05210=1064.977,-83.074,439.042,171.864,24.701,154.580
C05211=1064.983,-82.824,439.031,171.865,24.702,154.580
C05212=1064.990,-82.543,439.018,171.867,24.704,154.580
C05213=1064.997,-82.261,439.006,171.870,24.706,154.580
C05214=1065.004,-81.980,438.994,171.871,24.707,154.580
C05215=1065.012,-81.699,438.982,171.873,24.709,154.580
C05216=1065.017,-81.450,438.971,171.874,24.710,154.580
C05217=1065.024,-81.199,438.960,171.876,24.712,154.580
C05218=1065.030,-80.950,438.949,171.878,24.713,154.580
C05219=1065.037,-80.700,438.938,171.879,24.715,154.580
C05220=1065.042,-80.451,438.928,171.881,24.717,154.580
C05221=1065.048,-80.201,438.917,171.882,24.718,154.580
C05222=1065.054,-79.951,438.905,171.885,24.720,154.581
C05223=1065.061,-79.702,438.895,171.887,24.721,154.581
C05224=1065.067,-79.451,438.884,171.888,24.723,154.581
C05225=1065.073,-79.202,438.873,171.890,24.724,154.581
C05226=1065.079,-78.952,438.862,171.891,24.726,154.581
C05227=1065.085,-78.702,438.851,171.893,24.728,154.581
C05228=1065.091,-78.453,438.840,171.895,24.729,154.581
C05229=1065.097,-78.203,438.828,171.896,24.731,154.581
C05230=1065.103,-77.954,438.817,171.898,24.732,154.581
C05231=1065.110,-77.704,438.806,171.899,24.734,154.581
C05232=1065.115,-77.454,438.795,171.901,24.736,154.581
C05233=1065.121,-77.205,438.784,171.903,24.737,154.581
C05234=1065.127,-76.954,438.773,171.904,24.739,154.582
C05235=1065.134,-76.705,438.763,171.906,24.741,154.582
C05236=1065.140,-76.456,438.751,171.907,24.742,154.582
C05237=1065.146,-76.206,438.740,171.909,24.744,154.582
C05238=1065.153,-75.956,438.729,171.911,24.746,154.582
C05239=1065.158,-75.706,438.718,171.912,24.747,154.582
C05240=1065.164,-75.457,438.707,171.914,24.749,154.582
C05241=1065.171,-75.207,438.695,171.915,24.750,154.582
C05242=1065.176,-74.958,438.684,171.917,24.752,154.582
C05243=1065.183,-74.708,438.673,171.919,24.753,154.583
C05244=1065.188,-74.458,438.662,171.921,24.756,154.583
C05245=1065.195,-74.209,438.650,171.923,24.757,154.583
C05246=1065.201,-73.959,438.639,171.924,24.759,154.583
C05247=1065.207,-73.709,438.628,171.926,24.760,154.583
C05248=1065.213,-73.459,438.617,171.927,24.762,154.583
C05249=1065.220,-73.210,438.605,171.929,24.764,154.583
C05250=1065.225,-72.960,438.594,171.931,24.765,154.583
C05251=1065.230,-72.711,438.583,171.932,24.767,154.583
C05252=1065.237,-72.460,438.571,171.934,24.769,154.583
C05253=1065.243,-72.212,438.560,171.935,24.771,154.584
C05254=1065.249,-71.961,438.549,171.937,24.773,154.584
C05255=1065.254,-71.712,438.537,171.938,24.774,154.584
C05256=1065.261,-71.462,438.525,171.940,24.776,154.584
C05257=1065.266,-71.213,438.514,171.942,24.777,154.584
C05258=1065.273,-70.962,438.503,171.943,24.779,154.584
C05259=1065.279,-70.713,438.491,171.945,24.781,154.584
C05260=1065.284,-70.463,438.480,171.946,24.783,154.584
C05261=1065.290,-70.213,438.469,171.948,24.785,154.585
C05262=1065.297,-69.964,438.457,171.949,24.787,154.585
C05263=1065.303,-69.714,438.446,171.951,24.788,154.585
C05264=1065.309,-69.465,438.434,171.953,24.790,154.585
C05265=1065.314,-69.215,438.422,171.955,24.792,154.585
C05266=1065.321,-68.965,438.411,171.957,24.794,154.585
C05267=1065.327,-68.716,438.400,171.958,24.795,154.585
C05268=1065.333,-68.466,438.388,171.960,24.797,154.585
C05269=1065.339,-68.217,438.377,171.961,24.799,154.586
C05270=1065.345,-67.966,438.365,171.963,24.801,154.586
C05271=1065.351,-67.718,438.353,171.964,24.803,154.586
C05272=1065.357,-67.467,438.342,171.966,24.804,154.586
C05273=1065.363,-67.218,438.331,171.968,24.806,154.586
C05274=1065.369,-66.968,438.319,171.969,24.808,154.586
C05275=1065.374,-66.718,438.308,171.971,24.810,154.586
C05276=1065.382,-66.439,438.294,171.972,24.812,154.587
C05277=1065.388,-66.160,438.281,171.975,24.814,154.587
C05278=1065.396,-65.881,438.269,171.976,24.816,154.587
C05279=1065.402,-65.602,438.256,171.978,24.818,154.587
C05280=1065.407,-65.352,438.244,171.979,24.820,154.587
C05281=1065.414,-65.102,438.232,171.981,24.822,154.587
C05282=1065.420,-64.853,438.221,171.982,24.823,154.588
C05283=1065.426,-64.603,438.209,171.984,24.825,154.588
C05284=1065.432,-64.354,438.197,171.985,24.827,154.588
C05285=1065.438,-64.104,438.186,171.987,24.829,154.588
C05286=1065.445,-63.854,438.174,171.988,24.831,154.588
C05287=1065.450,-63.605,438.163,171.991,24.833,154.588
C05288=1065.456,-63.355,438.151,171.993,24.835,154.588
C05289=1065.462,-63.105,438.140,171.994,24.836,154.588
C05290=1065.469,-62.856,438.128,171.996,24.838,154.589
C05291=1065.475,-62.606,438.116,171.997,24.840,154.589
C05292=1065.480,-62.356,438.104,171.999,24.842,154.589
C05293=1065.487,-62.107,438.092,172.000,24.844,154.589
C05294=1065.493,-61.856,438.081,172.002,24.845,154.589
C05295=1065.499,-61.607,438.069,172.003,24.847,154.589
C05296=1065.505,-61.358,438.057,172.005,24.849,154.589
C05297=1065.511,-61.108,438.046,172.006,24.851,154.590
C05298=1065.517,-60.858,438.033,172.008,24.853,154.590
C05299=1065.524,-60.609,438.022,172.010,24.855,154.590
C05300=1065.529,-60.359,438.011,172.011,24.856,154.590
C05301=1065.536,-60.110,437.999,172.013,24.858,154.590
C05302=1065.542,-59.860,437.986,172.014,24.860,154.590
C05303=1065.548,-59.610,437.975,172.016,24.862,154.590
C05304=1065.554,-59.361,437.963,172.017,24.864,154.591
C05305=1065.560,-59.111,437.951,172.019,24.866,154.591
C05306=1065.567,-58.861,437.940,172.020,24.868,154.591
C05307=1065.573,-58.612,437.928,172.022,24.870,154.591
C05308=1065.579,-58.362,437.915,172.024,24.872,154.591
C05309=1065.585,-58.112,437.903,172.026,24.874,154.591
C05310=1065.591,-57.863,437.893,172.027,24.875,154.592
C05311=1065.597,-57.613,437.880,172.029,24.877,154.592
C05312=1065.603,-57.363,437.868,172.031,24.879,154.592
C05313=1065.610,-57.114,437.856,172.032,24.881,154.592
C05314=1065.615,-56.864,437.845,172.034,24.883,154.592
C05315=1065.622,-56.614,437.833,172.035,24.885,154.592
C05316=1065.628,-56.365,437.821,172.037,24.887,154.593
C05317=1065.634,-56.115,437.808,172.038,24.889,154.593
C05318=1065.640,-55.866,437.797,172.040,24.890,154.593
C05319=1065.646,-55.616,437.785,172.041,24.892,154.593
C05320=1065.653,-55.366,437.773,172.043,24.894,154.593
C05321=1065.659,-55.116,437.761,172.044,24.896,154.593
C05322=1065.665,-54.867,437.749,172.046,24.898,154.594
C05323=1065.671,-54.618,437.737,172.047,24.900,154.594
C05324=1065.678,-54.368,437.725,172.049,24.902,154.594
C05325=1065.683,-54.118,437.713,172.051,24.904,154.594
C05326=1065.690,-53.869,437.701,172.052,24.905,154.594
C05327=1065.696,-53.619,437.689,172.054,24.907,154.594
C05328=1065.702,-53.369,437.677,172.056,24.909,154.594
C05329=1065.709,-53.120,437.665,172.058,24.912,154.595
C05330=1065.715,-52.870,437.652,172.059,24.914,154.595
C05331=1065.721,-52.620,437.641,172.061,24.915,154.595
C05332=1065.727,-52.371,437.629,172.062,24.917,154.595
C05333=1065.733,-52.121,437.617,172.064,24.919,154.595
C05334=1065.740,-51.871,437.605,172.065,24.921,154.595
C05335=1065.745,-51.621,437.592,172.067,24.923,154.596
C05336=1065.752,-51.372,437.580,172.068,24.925,154.596
C05337=1065.758,-51.123,437.569,172.070,24.927,154.596
C05338=1065.764,-50.873,437.556,172.071,24.929,154.596
C05339=1065.771,-50.624,437.544,172.073,24.931,154.596
C05340=1065.777,-50.345,437.531,172.074,24.933,154.596
C05341=1065.784,-50.068,437.517,172.077,24.935,154.597
C05342=1065.791,-49.789,437.503,172.078,24.937,154.597
C05343=1065.798,-49.511,437.489,172.080,24.940,154.597
C05344=1065.804,-49.263,437.477,172.081,24.941,154.597
C05345=1065.810,-49.013,437.465,172.083,24.944,154.597
C05346=1065.816,-48.763,437.452,172.084,24.946,154.598
C05347=1065.822,-48.513,437.440,172.086,24.948,154.598
C05348=1065.828,-48.264,437.428,172.087,24.950,154.598
C05349=1065.833,-48.014,437.416,172.089,24.952,154.598
C05350=1065.839,-47.764,437.403,172.090,24.954,154.598
C05351=1065.846,-47.515,437.391,172.092,24.956,154.599
C05352=1065.852,-47.265,437.379,172.094,24.958,154.599
C05353=1065.857,-47.016,437.366,172.096,24.960,154.599
C05354=1065.864,-46.766,437.354,172.097,24.963,154.599
C05355=1065.870,-46.516,437.342,172.099,24.964,154.599
C05356=1065.876,-46.266,437.329,172.100,24.966,154.599
C05357=1065.882,-46.016,437.317,172.102,24.969,154.600
C05358=1065.889,-45.767,437.304,172.103,24.970,154.600
C05359=1065.894,-45.518,437.292,172.105,24.973,154.600
C05360=1065.900,-45.268,437.279,172.106,24.975,154.600
C05361=1065.906,-45.019,437.267,172.108,24.977,154.601
C05362=1065.912,-44.769,437.255,172.109,24.979,154.601
C05363=1065.918,-44.519,437.242,172.111,24.981,154.601
C05364=1065.924,-44.269,437.230,172.112,24.983,154.601
C05365=1065.931,-44.020,437.217,172.113,24.985,154.601
C05366=1065.937,-43.770,437.204,172.115,24.987,154.602
C05367=1065.942,-43.521,437.192,172.117,24.989,154.602
C05368=1065.948,-43.271,437.180,172.118,24.991,154.602
C05369=1065.955,-43.022,437.168,172.120,24.993,154.602
C05370=1065.961,-42.772,437.155,172.121,24.995,154.602
C05371=1065.967,-42.523,437.142,172.123,24.997,154.603
C05372=1065.973,-42.273,437.129,172.124,25.000,154.603
C05373=1065.980,-42.023,437.117,172.126,25.001,154.603
C05374=1065.985,-41.773,437.105,172.127,25.004,154.603
C05375=1065.992,-41.524,437.092,172.129,25.006,154.603
C05376=1065.998,-41.274,437.079,172.131,25.008,154.604
C05377=1066.004,-41.025,437.067,172.132,25.010,154.604
C05378=1066.010,-40.775,437.055,172.134,25.012,154.604
C05379=1066.016,-40.526,437.042,172.135,25.014,154.604
C05380=1066.022,-40.276,437.029,172.137,25.017,154.604
C05381=1066.028,-40.026,437.017,172.138,25.018,154.605
C05382=1066.034,-39.777,437.005,172.140,25.021,154.605
C05383=1066.040,-39.527,436.991,172.141,25.023,154.605
C05384=1066.046,-39.278,436.979,172.143,25.025,154.605
C05385=1066.052,-39.028,436.966,172.144,25.027,154.605
C05386=1066.059,-38.779,436.954,172.146,25.029,154.606
C05387=1066.065,-38.529,436.941,172.147,25.031,154.606
C05388=1066.071,-38.279,436.928,172.149,25.033,154.606
C05389=1066.077,-38.030,436.915,172.150,25.036,154.606
C05390=1066.083,-37.780,436.903,172.152,25.038,154.607
C05391=1066.089,-37.530,436.890,172.153,25.040,154.607
C05392=1066.095,-37.281,436.877,172.155,25.042,154.607
C05393=1066.101,-37.031,436.864,172.156,25.045,154.607
C05394=1066.107,-36.782,436.851,172.158,25.046,154.607
C05395=1066.113,-36.532,436.838,172.159,25.049,154.608
C05396=1066.119,-36.282,436.826,172.160,25.051,154.608
C05397=1066.125,-36.033,436.813,172.162,25.053,154.608
C05398=1066.131,-35.783,436.800,172.163,25.055,154.608
C05399=1066.137,-35.534,436.787,172.165,25.058,154.609
C05400=1066.143,-35.284,436.775,172.166,25.059,154.609
C05401=1066.149,-35.034,436.762,172.168,25.062,154.609
C05402=1066.155,-34.785,436.749,172.169,25.064,154.609
C05403=1066.161,-34.535,436.736,172.172,25.066,154.609
C05404=1066.168,-34.258,436.721,172.173,25.069,154.610
C05405=1066.174,-33.980,436.707,172.175,25.071,154.610
C05406=1066.181,-33.702,436.692,172.176,25.073,154.610
C05407=1066.188,-33.425,436.678,172.178,25.076,154.610
C05408=1066.194,-33.175,436.665,172.180,25.078,154.611
C05409=1066.200,-32.925,436.652,172.181,25.081,154.611
C05410=1066.206,-32.676,436.639,172.183,25.083,154.611
C05411=1066.212,-32.426,436.627,172.184,25.085,154.611
C05412=1066.219,-32.177,436.613,172.186,25.087,154.612
C05413=1066.224,-31.927,436.601,172.187,25.090,154.612
C05414=1066.231,-31.678,436.587,172.189,25.092,154.612
C05415=1066.237,-31.428,436.575,172.190,25.094,154.612
C05416=1066.243,-31.179,436.562,172.191,25.096,154.613
C05417=1066.249,-30.930,436.548,172.193,25.099,154.613
C05418=1066.255,-30.680,436.536,172.194,25.100,154.613
C05419=1066.261,-30.430,436.523,172.196,25.103,154.613
C05420=1066.267,-30.180,436.510,172.197,25.105,154.614
C05421=1066.273,-29.931,436.496,172.199,25.107,154.614
C05422=1066.278,-29.681,436.484,172.200,25.109,154.614
C05423=1066.285,-29.432,436.470,172.202,25.112,154.614
C05424=1066.291,-29.182,436.457,172.203,25.114,154.615
C05425=1066.297,-28.932,436.444,172.205,25.116,154.615
C05426=1066.304,-28.683,436.431,172.206,25.118,154.615
C05427=1066.310,-28.433,436.418,172.208,25.121,154.615
C05428=1066.316,-28.184,436.405,172.209,25.123,154.615
C05429=1066.322,-27.934,436.392,172.210,25.125,154.616
C05430=1066.328,-27.685,436.378,172.212,25.127,154.616
C05431=1066.334,-27.435,436.366,172.213,25.129,154.616
C05432=1066.340,-27.186,436.353,172.215,25.132,154.616
C05433=1066.347,-26.936,436.339,172.216,25.134,154.617
C05434=1066.352,-26.686,436.326,172.218,25.136,154.617
C05435=1066.358,-26.436,436.313,172.219,25.138,154.617
C05436=1066.365,-26.187,436.299,172.221,25.141,154.617
C05437=1066.371,-25.937,436.287,172.223,25.143,154.618
C05438=1066.376,-25.688,436.273,172.225,25.146,154.618
C05439=1066.382,-25.438,436.260,172.226,25.148,154.618
C05440=1066.388,-25.189,436.246,172.227,25.150,154.618
C05441=1066.394,-24.939,436.233,172.229,25.153,154.619
C05442=1066.400,-24.690,436.220,172.230,25.155,154.619
C05443=1066.407,-24.440,436.206,172.232,25.157,154.619
C05444=1066.413,-24.190,436.193,172.233,25.159,154.619
C05445=1066.418,-23.941,436.179,172.235,25.162,154.620
C05446=1066.424,-23.691,436.167,172.236,25.164,154.620
C05447=1066.431,-23.442,436.153,172.238,25.166,154.620
C05448=1066.436,-23.192,436.140,172.239,25.169,154.620
C05449=1066.442,-22.943,436.126,172.240,25.171,154.621
C05450=1066.448,-22.694,436.113,172.242,25.173,154.621
C05451=1066.454,-22.443,436.099,172.243,25.176,154.621
C05452=1066.460,-22.193,436.086,172.245,25.178,154.622
C05453=1066.467,-21.944,436.073,172.246,25.181,154.622
